KUKA KRL program: MyProgram_249().src

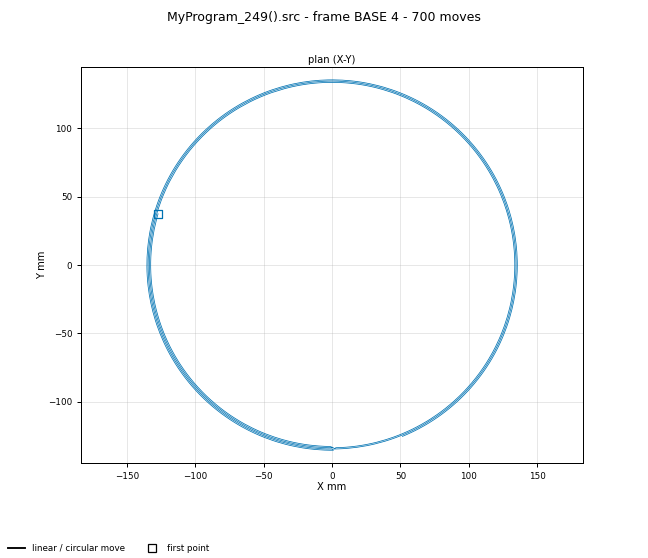
[picture p0: tool path of MyProgram_249().src in frame BASE 4, 700 of 700 moves have a stored position in this frame; points joined in program order, loops and branches not executed]
&ACCESS RVP
&REL 1
&PARAM TEMPLATE = C:\KRC\Roboter\Template\vorgabe
&PARAM EDITMASK = *
DEF MyProgram_249()
; ---- Setting reference (Base) ----
$BASE = BASE_DATA[4]

; --------------------------
; ---- Setting tool (TCP) ----
$TOOL = TOOL_DATA[3]
; --------------------------

$VEL.CP = VEL_APROX_PRINT
Startdeposition()
$VEL.CP = VEL_PRINT
LIN {X -127.2859,Y 37.4504,Z 164,A 163.9106,B 12.714,C 0.0045,E1 12.5602,E2 286.2896} C_DIS
LIN {X -128.1717,Y 34.2964,Z 164,A 165.3545,B 12.714,C 0.0079,E1 12.5591,E2 284.844} C_DIS
LIN {X -130.1138,Y 25.9783,Z 164,A 168.8195,B 12.714,C 0.0239,E1 12.557,E2 281.4101} C_DIS
LIN {X -131.4651,Y 17.9356,Z 164,A 172.8382,B 12.714,C 0.0228,E1 12.5551,E2 277.3369} C_DIS
LIN {X -131.9904,Y 13.5371,Z 164,A 174.6216,B 12.714,C 0.0315,E1 12.5546,E2 275.5713} C_DIS
LIN {X -132.3145,Y 9.8588,Z 164,A 176.2918,B 12.714,C 0.0344,E1 12.5542,E2 273.8938} C_DIS
LIN {X -132.5525,Y 5.8863,Z 164,A 178.0814,B 12.714,C 0.0379,E1 12.5539,E2 272.0978} C_DIS
LIN {X -132.6635,Y 2.1671,Z 164,A 179.6659,B 12.714,C 0.0432,E1 12.5539,E2 270.5176} C_DIS
LIN {X -132.6704,Y -1.7531,Z 164,A -178.5856,B 12.714,C 0.0469,E1 12.5539,E2 268.7644} C_DIS
LIN {X -132.5551,Y -5.8195,Z 164,A -176.8371,B 12.714,C 0.0523,E1 12.554,E2 267.0189} C_DIS
LIN {X -132.3464,Y -9.4225,Z 164,A -175.2437,B 12.714,C 0.0561,E1 12.5543,E2 265.423} C_DIS
LIN {X -132.026,Y -13.1779,Z 164,A -173.5549,B 12.7139,C 0.0595,E1 12.5548,E2 263.7286} C_DIS
LIN {X -131.5827,Y -17.0384,Z 164,A -171.2367,B 12.7139,C 0.0494,E1 12.5556,E2 261.3351} C_DIS
LIN {X -130.7769,Y -22.4052,Z 164,A -169.5669,B 12.7139,C 0.072,E1 12.5564,E2 259.749} C_DIS
LIN {X -129.5394,Y -28.7106,Z 164,A -166.6985,B 12.7138,C 0.0779,E1 12.558,E2 256.8722} C_DIS
LIN {X -128.5013,Y -33.0423,Z 164,A -164.2137,B 12.7138,C 0.0701,E1 12.5597,E2 254.3216} C_DIS
LIN {X -127.2066,Y -37.7213,Z 164,A -162.6596,B 12.7138,C 0.0888,E1 12.5609,E2 252.8349} C_DIS
LIN {X -125.9532,Y -41.7138,Z 164,A -160.9153,B 12.7137,C 0.0954,E1 12.5623,E2 251.0997} C_DIS
LIN {X -124.788,Y -45.0792,Z 164,A -159.3157,B 12.7137,C 0.0982,E1 12.5638,E2 249.4941} C_DIS
LIN {X -123.3299,Y -48.933,Z 164,A -157.4471,B 12.7137,C 0.1009,E1 12.5657,E2 247.6164} C_DIS
LIN {X -122.0827,Y -51.9667,Z 164,A -156.1315,B 12.7136,C 0.1071,E1 12.5671,E2 246.3141} C_DIS
LIN {X -120.6653,Y -55.1756,Z 164,A -154.4483,B 12.7136,C 0.1071,E1 12.5691,E2 244.6119} C_DIS
LIN {X -118.5377,Y -59.6103,Z 164,A -152.3885,B 12.7136,C 0.1142,E1 12.5716,E2 242.5616} C_DIS
LIN {X -116.8408,Y -62.8722,Z 164,A -150.792,B 12.7135,C 0.1181,E1 12.5737,E2 240.9653} C_DIS
LIN {X -114.9119,Y -66.3322,Z 164,A -148.9965,B 12.7135,C 0.1204,E1 12.5762,E2 239.1609} C_DIS
LIN {X -112.7429,Y -69.9553,Z 164,A -146.8726,B 12.7135,C 0.1177,E1 12.5793,E2 237.0019} C_DIS
LIN {X -110.8171,Y -72.9675,Z 164,A -145.2284,B 12.7135,C 0.119,E1 12.5819,E2 235.3465} C_DIS
LIN {X -108.5489,Y -76.3012,Z 164,A -143.8692,B 12.7133,C 0.1323,E1 12.584,E2 234.0348} C_DIS
LIN {X -106.1417,Y -79.6164,Z 164,A -142.0172,B 12.7133,C 0.1344,E1 12.5871,E2 232.1738} C_DIS
LIN {X -103.4343,Y -83.1029,Z 164,A -140.1059,B 12.7133,C 0.1386,E1 12.5904,E2 230.2631} C_DIS
LIN {X -101.023,Y -86.0177,Z 164,A -138.0843,B 12.7133,C 0.1327,E1 12.5941,E2 228.1952} C_DIS
LIN {X -98.2832,Y -89.135,Z 164,A -136.5931,B 12.7133,C 0.1438,E1 12.5968,E2 226.7415} C_DIS
LIN {X -95.0015,Y -92.6258,Z 164,A -134.5379,B 12.7132,C 0.1484,E1 12.6008,E2 224.6891} C_DIS
LIN {X -91.8567,Y -95.7449,Z 164,A -132.7035,B 12.7132,C 0.1541,E1 12.6044,E2 222.865} C_DIS
LIN {X -88.8171,Y -98.5716,Z 164,A -130.8078,B 12.7131,C 0.155,E1 12.6084,E2 220.9575} C_DIS
LIN {X -83.7542,Y -102.9072,Z 164,A -127.8819,B 12.7131,C 0.1591,E1 12.6147,E2 218.0268} C_DIS
LIN {X -80.3922,Y -105.5549,Z 164,A -126.3364,B 12.7129,C 0.1698,E1 12.618,E2 216.5186} C_DIS
LIN {X -77.3944,Y -107.7723,Z 164,A -124.7502,B 12.7129,C 0.173,E1 12.6215,E2 214.9358} C_DIS
LIN {X -74.3027,Y -109.9264,Z 164,A -122.8693,B 12.7129,C 0.1692,E1 12.6259,E2 213.0246} C_DIS
LIN {X -71.2377,Y -111.9375,Z 164,A -121.027,B 12.7129,C 0.1651,E1 12.6303,E2 211.151} C_DIS
LIN {X -66.9659,Y -114.544,Z 164,A -119.1475,B 12.7129,C 0.1752,E1 12.6348,E2 209.3062} C_DIS
LIN {X -63.868,Y -116.2999,Z 164,A -117.7538,B 12.7128,C 0.1809,E1 12.6381,E2 207.9301} C_DIS
LIN {X -60.867,Y -117.8979,Z 164,A -116.1634,B 12.7128,C 0.1797,E1 12.6421,E2 206.3251} C_DIS
LIN {X -58.2643,Y -119.2043,Z 164,A -114.7229,B 12.7128,C 0.1765,E1 12.6457,E2 204.8623} C_DIS
LIN {X -54.5493,Y -120.9492,Z 164,A -113.2139,B 12.7127,C 0.1852,E1 12.6495,E2 203.3854} C_DIS
LIN {X -51.4956,Y -122.2805,Z 164,A -111.5729,B 12.7127,C 0.1815,E1 12.6538,E2 201.7199} C_DIS
LIN {X -48.452,Y -123.5182,Z 164,A -110.1328,B 12.7127,C 0.1824,E1 12.6575,E2 200.2771} C_DIS
LIN {X -44.8785,Y -124.8604,Z 164,A -108.5366,B 12.7127,C 0.1852,E1 12.6617,E2 198.6871} C_DIS
LIN {X -42.0608,Y -125.8376,Z 164,A -107.0295,B 12.7127,C 0.1805,E1 12.6657,E2 197.1532} C_DIS
LIN {X -36.4597,Y -127.5753,Z 164,A -104.6656,B 12.7127,C 0.1868,E1 12.672,E2 194.8096} C_DIS
LIN {X -31.6264,Y -128.8576,Z 164,A -102.4818,B 12.7127,C 0.1874,E1 12.6779,E2 192.6224} C_DIS
LIN {X -27.87,Y -129.7209,Z 164,A -100.846,B 12.7127,C 0.189,E1 12.6824,E2 190.9897} C_DIS
LIN {X -23.7795,Y -130.5333,Z 164,A -99.0245,B 12.7127,C 0.1892,E1 12.6874,E2 189.1652} C_DIS
LIN {X -19.9907,Y -131.1668,Z 164,A -97.3285,B 12.7127,C 0.1888,E1 12.6921,E2 187.4642} C_DIS
LIN {X -16.2833,Y -131.6793,Z 164,A -95.708,B 12.7127,C 0.1891,E1 12.6966,E2 185.8426} C_DIS
LIN {X -12.7821,Y -132.064,Z 164,A -94.3224,B 12.7126,C 0.1929,E1 12.7004,E2 184.4731} C_DIS
LIN {X -9.6689,Y -132.3284,Z 164,A -92.921,B 12.7126,C 0.1917,E1 12.7043,E2 183.0647} C_DIS
LIN {X -5.4853,Y -132.5681,Z 164,A -91.0911,B 12.7126,C 0.1911,E1 12.7094,E2 181.2315} C_DIS
LIN {X -1.4506,Y -132.6753,Z 164,A -89.2488,B 12.7126,C 0.1883,E1 12.7146,E2 179.3764} C_DIS
LIN {X -1.4506,Y -132.6753,Z 164,A -89.2488,B 12.7126,C 0.1883,E1 12.7146,E2 179.3764} C_DIS
Enddeposition()
LIN {X 0.969,Y -133.5975,Z 164,A -88.8954,B 12.4309,C 0.2318,E1 12.434,E2 179.2272} C_DIS
Startdeposition()
$VEL.CP = VEL_PRINT
LIN {X -2.4265,Y -133.579,Z 164,A -90.4296,B 12.4309,C 0.2339,E1 12.4297,E2 180.7716} C_DIS
LIN {X -6.5842,Y -133.4385,Z 164,A -92.1314,B 12.4309,C 0.2318,E1 12.425,E2 182.4641} C_DIS
LIN {X -10.1796,Y -133.2132,Z 164,A -93.6549,B 12.4309,C 0.2312,E1 12.4207,E2 183.9856} C_DIS
LIN {X -14.0414,Y -132.8611,Z 164,A -95.3566,B 12.4309,C 0.2319,E1 12.416,E2 185.6927} C_DIS
LIN {X -17.9058,Y -132.3965,Z 164,A -97.0831,B 12.4309,C 0.233,E1 12.4112,E2 187.4267} C_DIS
LIN {X -21.716,Y -131.8242,Z 164,A -98.6443,B 12.4309,C 0.2301,E1 12.4069,E2 188.9773} C_DIS
LIN {X -24.9459,Y -131.2511,Z 164,A -100.0743,B 12.4309,C 0.2301,E1 12.403,E2 190.4105} C_DIS
LIN {X -28.3703,Y -130.5537,Z 164,A -101.5641,B 12.4309,C 0.2292,E1 12.3989,E2 191.8996} C_DIS
LIN {X -32.1236,Y -129.6833,Z 164,A -103.5588,B 12.4309,C 0.237,E1 12.3934,E2 193.9362} C_DIS
LIN {X -35.422,Y -128.8205,Z 164,A -104.7421,B 12.4309,C 0.229,E1 12.3903,E2 195.086} C_DIS
LIN {X -39.156,Y -127.7337,Z 164,A -106.311,B 12.431,C 0.2253,E1 12.3861,E2 196.643} C_DIS
LIN {X -42.2612,Y -126.7402,Z 164,A -107.7812,B 12.431,C 0.226,E1 12.3822,E2 198.1221} C_DIS
LIN {X -45.5289,Y -125.6035,Z 164,A -109.2648,B 12.431,C 0.2247,E1 12.3783,E2 199.6059} C_DIS
LIN {X -48.8747,Y -124.3406,Z 164,A -110.7775,B 12.431,C 0.2228,E1 12.3743,E2 201.1161} C_DIS
LIN {X -52.0639,Y -123.0398,Z 164,A -112.2452,B 12.4311,C 0.221,E1 12.3705,E2 202.5827} C_DIS
LIN {X -54.7996,Y -121.8447,Z 164,A -113.5516,B 12.4311,C 0.2203,E1 12.3672,E2 203.8922} C_DIS
LIN {X -58.0083,Y -120.3507,Z 164,A -115.2414,B 12.4311,C 0.2228,E1 12.3629,E2 205.6027} C_DIS
LIN {X -61.7986,Y -118.4487,Z 164,A -116.9737,B 12.4311,C 0.2184,E1 12.3586,E2 207.3245} C_DIS
LIN {X -65.64,Y -116.3658,Z 164,A -118.894,B 12.4311,C 0.2171,E1 12.3539,E2 209.2502} C_DIS
LIN {X -70.4553,Y -113.5145,Z 164,A -121.2134,B 12.4313,C 0.2118,E1 12.3484,E2 211.5595} C_DIS
LIN {X -73.3669,Y -111.6552,Z 164,A -122.786,B 12.4313,C 0.2118,E1 12.3447,E2 213.1428} C_DIS
LIN {X -77.4171,Y -108.8866,Z 164,A -124.79,B 12.4313,C 0.206,E1 12.3401,E2 215.1342} C_DIS
LIN {X -80.6674,Y -106.5007,Z 164,A -126.4,B 12.4315,C 0.2002,E1 12.3365,E2 216.7293} C_DIS
LIN {X -83.028,Y -104.6707,Z 164,A -128.3488,B 12.4312,C 0.2141,E1 12.3321,E2 218.7582} C_DIS
LIN {X -86.3499,Y -101.9476,Z 164,A -129.6511,B 12.4315,C 0.1979,E1 12.3294,E2 219.995} C_DIS
LIN {X -88.928,Y -99.7068,Z 164,A -131.2517,B 12.4315,C 0.1984,E1 12.326,E2 221.6115} C_DIS
LIN {X -92.0866,Y -96.7973,Z 164,A -133.0736,B 12.4315,C 0.1944,E1 12.3223,E2 223.4302} C_DIS
LIN {X -94.9521,Y -93.9879,Z 164,A -134.8716,B 12.4315,C 0.1927,E1 12.3187,E2 225.2367} C_DIS
LIN {X -97.949,Y -90.8604,Z 164,A -137.1822,B 12.4315,C 0.1996,E1 12.3142,E2 227.6007} C_DIS
LIN {X -100.953,Y -87.5114,Z 164,A -138.4296,B 12.4318,C 0.1794,E1 12.3121,E2 228.7653} C_DIS
LIN {X -102.7055,Y -85.4473,Z 164,A -139.8951,B 12.4318,C 0.184,E1 12.3094,E2 230.2669} C_DIS
LIN {X -105.5735,Y -81.8768,Z 164,A -141.7703,B 12.4318,C 0.1775,E1 12.3062,E2 232.1302} C_DIS
LIN {X -107.9313,Y -78.7438,Z 164,A -143.5646,B 12.4318,C 0.1763,E1 12.3032,E2 233.9371} C_DIS
LIN {X -110.9733,Y -74.3946,Z 164,A -145.7108,B 12.4319,C 0.1679,E1 12.2998,E2 236.0663} C_DIS
LIN {X -113.4173,Y -70.6123,Z 164,A -147.7572,B 12.4319,C 0.1658,E1 12.2967,E2 238.1251} C_DIS
LIN {X -115.5704,Y -67.0303,Z 164,A -149.5797,B 12.432,C 0.1621,E1 12.2941,E2 239.95} C_DIS
LIN {X -117.5621,Y -63.4729,Z 164,A -151.3707,B 12.432,C 0.1586,E1 12.2917,E2 241.7448} C_DIS
LIN {X -119.4403,Y -59.8644,Z 164,A -153.3097,B 12.432,C 0.1586,E1 12.2892,E2 243.7057} C_DIS
LIN {X -121.6776,Y -55.1732,Z 164,A -155.4943,B 12.4321,C 0.1517,E1 12.2866,E2 245.8832} C_DIS
LIN {X -123.4205,Y -51.1523,Z 164,A -157.1832,B 12.4322,C 0.1423,E1 12.2848,E2 247.5477} C_DIS
LIN {X -124.8044,Y -47.6815,Z 164,A -158.798,B 12.4322,C 0.1382,E1 12.2832,E2 249.1627} C_DIS
LIN {X -125.8056,Y -44.9683,Z 164,A -160.0935,B 12.4323,C 0.136,E1 12.2819,E2 250.4636} C_DIS
LIN {X -127.0792,Y -41.235,Z 164,A -161.8357,B 12.4323,C 0.1325,E1 12.2804,E2 252.2104} C_DIS
LIN {X -128.2024,Y -37.5929,Z 164,A -164.0108,B 12.4323,C 0.1402,E1 12.2786,E2 254.4481} C_DIS
LIN {X -129.4444,Y -33.0647,Z 164,A -165.5735,B 12.4324,C 0.1243,E1 12.2776,E2 255.9555} C_DIS
LIN {X -130.6401,Y -27.9703,Z 164,A -168.3192,B 12.4324,C 0.1291,E1 12.2759,E2 258.7584} C_DIS
LIN {X -131.5391,Y -23.3797,Z 164,A -169.7929,B 12.4326,C 0.1114,E1 12.2752,E2 260.1671} C_DIS
LIN {X -132.3855,Y -17.9896,Z 164,A -172.1913,B 12.4326,C 0.1059,E1 12.2742,E2 262.5701} C_DIS
LIN {X -132.8479,Y -14.1632,Z 164,A -173.8147,B 12.4326,C 0.1003,E1 12.2737,E2 264.1883} C_DIS
LIN {X -133.2229,Y -10.0464,Z 164,A -175.6612,B 12.4326,C 0.0968,E1 12.2732,E2 266.0417} C_DIS
LIN {X -133.4376,Y -6.6024,Z 164,A -177.1199,B 12.4327,C 0.0919,E1 12.273,E2 267.4962} C_DIS
LIN {X -133.5742,Y -2.7138,Z 164,A -178.874,B 12.4327,C 0.0889,E1 12.2729,E2 269.2587} C_DIS
LIN {X -133.5972,Y 1.0787,Z 164,A 179.4492,B 12.4327,C 0.0853,E1 12.2729,E2 270.9397} C_DIS
LIN {X -133.5003,Y 5.1826,Z 164,A 177.7929,B 12.4328,C 0.0777,E1 12.273,E2 272.5816} C_DIS
LIN {X -133.328,Y 8.5399,Z 164,A 176.3503,B 12.4328,C 0.0734,E1 12.2732,E2 274.0227} C_DIS
LIN {X -133.0541,Y 12.092,Z 164,A 174.658,B 12.4328,C 0.0726,E1 12.2736,E2 275.7329} C_DIS
LIN {X -132.6486,Y 15.9224,Z 164,A 173.0231,B 12.4328,C 0.0673,E1 12.2741,E2 277.3637} C_DIS
LIN {X -131.3055,Y 24.6614,Z 164,A 169.4185,B 12.4329,C 0.052,E1 12.2757,E2 280.9419} C_DIS
LIN {X -130.3282,Y 29.3907,Z 164,A 166.9317,B 12.4329,C 0.0553,E1 12.2772,E2 283.4754} C_DIS
LIN {X -129.1549,Y 34.1785,Z 164,A 164.9442,B 12.4329,C 0.0464,E1 12.2785,E2 285.4455} C_DIS
LIN {X -128.1565,Y 37.7498,Z 164,A 163.4061,B 12.4329,C 0.0406,E1 12.2797,E2 286.9755} C_DIS
LIN {X -127.1567,Y 40.9924,Z 164,A 161.9634,B 12.4329,C 0.0362,E1 12.2809,E2 288.415} C_DIS
LIN {X -126.1016,Y 44.1317,Z 164,A 160.5161,B 12.433,C 0.0328,E1 12.2822,E2 289.8638} C_DIS
LIN {X -124.9839,Y 47.204,Z 164,A 159.0732,B 12.433,C 0.0298,E1 12.2836,E2 291.3099} C_DIS
LIN {X -123.7939,Y 50.2418,Z 164,A 157.6003,B 12.433,C 0.0275,E1 12.2852,E2 292.7898} C_DIS
LIN {X -121.5872,Y 55.3731,Z 164,A 155.2739,B 12.433,C 0.0194,E1 12.2878,E2 295.1052} C_DIS
LIN {X -120.0819,Y 58.5641,Z 164,A 153.5082,B 12.433,C 0.021,E1 12.2899,E2 296.8989} C_DIS
LIN {X -118.5664,Y 61.5743,Z 164,A 152.1424,B 12.433,C 0.0154,E1 12.2917,E2 298.2536} C_DIS
LIN {X -115.5947,Y 66.9882,Z 164,A 149.6992,B 12.433,C 0.0038,E1 12.295,E2 300.6695} C_DIS
LIN {X -114.4253,Y 68.9671,Z 164,A 147.98,B 12.433,C 0.0179,E1 12.2976,E2 302.4736} C_DIS
LIN {X -111.8785,Y 73.0265,Z 164,A 146.4944,B 12.433,C -0.0003,E1 12.2997,E2 303.8902} C_DIS
LIN {X -109.7337,Y 76.2109,Z 164,A 144.6442,B 12.433,C 0.0003,E1 12.3027,E2 305.7623} C_DIS
LIN {X -106.848,Y 80.2072,Z 164,A 142.5669,B 12.433,C -0.0057,E1 12.3061,E2 307.8329} C_DIS
LIN {X -104.0301,Y 83.829,Z 164,A 140.6438,B 12.433,C -0.0114,E1 12.3094,E2 309.7484} C_DIS
LIN {X -101.3278,Y 87.0763,Z 164,A 138.79,B 12.433,C -0.0146,E1 12.3128,E2 311.6051} C_DIS
LIN {X -98.5378,Y 90.2216,Z 164,A 136.94,B 12.433,C -0.0176,E1 12.3162,E2 313.4587} C_DIS
LIN {X -95.3819,Y 93.5514,Z 164,A 135.009,B 12.433,C -0.0227,E1 12.3199,E2 315.3831} C_DIS
LIN {X -92.2253,Y 96.6647,Z 164,A 133.0772,B 12.433,C -0.026,E1 12.3238,E2 317.3164} C_DIS
LIN {X -88.9304,Y 99.7047,Z 164,A 131.14,B 12.433,C -0.0296,E1 12.3278,E2 319.2533} C_DIS
LIN {X -85.6216,Y 102.5603,Z 164,A 129.2397,B 12.433,C -0.0327,E1 12.3319,E2 321.1546} C_DIS
LIN {X -82.2236,Y 105.3043,Z 164,A 127.3172,B 12.433,C -0.0351,E1 12.3361,E2 323.0809} C_DIS
LIN {X -78.5614,Y 108.0635,Z 164,A 125.3608,B 12.433,C -0.039,E1 12.3405,E2 325.0341} C_DIS
LIN {X -74.9376,Y 110.6071,Z 164,A 123.4511,B 12.433,C -0.042,E1 12.3449,E2 326.9432} C_DIS
LIN {X -71.3158,Y 112.9762,Z 164,A 121.6079,B 12.433,C -0.0454,E1 12.3492,E2 328.7831} C_DIS
LIN {X -67.6566,Y 115.2049,Z 164,A 119.7538,B 12.433,C -0.0479,E1 12.3536,E2 330.6373} C_DIS
LIN {X -60.2805,Y 119.2285,Z 164,A 116.1931,B 12.433,C -0.0542,E1 12.3624,E2 334.1897} C_DIS
LIN {X -56.5162,Y 121.0587,Z 164,A 113.7895,B 12.433,C -0.042,E1 12.3686,E2 336.6628} C_DIS
LIN {X -52.0532,Y 123.0443,Z 164,A 112.3832,B 12.4329,C -0.0611,E1 12.372,E2 337.9868} C_DIS
LIN {X -48.3185,Y 124.5568,Z 164,A 110.4886,B 12.4329,C -0.0591,E1 12.377,E2 339.8996} C_DIS
LIN {X -44.2124,Y 126.0737,Z 164,A 108.5419,B 12.4329,C -0.0594,E1 12.3821,E2 341.853} C_DIS
LIN {X -34.5806,Y 129.0477,Z 164,A 104.5946,B 12.4329,C -0.0726,E1 12.3925,E2 345.7527} C_DIS
LIN {X -29.4838,Y 130.3069,Z 164,A 101.4239,B 12.4329,C -0.0517,E1 12.4014,E2 349.0296} C_DIS
LIN {X -24.4604,Y 131.3439,Z 164,A 99.9031,B 12.4329,C -0.0697,E1 12.4054,E2 350.4697} C_DIS
LIN {X -21.7381,Y 131.8205,Z 164,A 98.642,B 12.4329,C -0.0685,E1 12.4089,E2 351.7389} C_DIS
LIN {X -17.7944,Y 132.4111,Z 164,A 96.9364,B 12.4329,C -0.0695,E1 12.4136,E2 353.443} C_DIS
LIN {X -14.2596,Y 132.8376,Z 164,A 95.4026,B 12.4329,C -0.0699,E1 12.4178,E2 354.9767} C_DIS
LIN {X -9.9853,Y 133.2274,Z 164,A 93.5465,B 12.4329,C -0.0701,E1 12.423,E2 356.8335} C_DIS
LIN {X -5.909,Y 133.472,Z 164,A 91.7239,B 12.4329,C -0.0687,E1 12.4281,E2 358.6637} C_DIS
LIN {X -2.1617,Y 133.5834,Z 164,A 90.2016,B 12.4329,C -0.0711,E1 12.4323,E2 360.1751} C_DIS
LIN {X 1.581,Y 133.5931,Z 164,A 88.5163,B 12.4329,C -0.0691,E1 12.437,E2 361.8691} C_DIS
LIN {X 5.7626,Y 133.4777,Z 164,A 86.718,B 12.4329,C -0.0689,E1 12.4421,E2 363.6671} C_DIS
LIN {X 9.8231,Y 133.2392,Z 164,A 85.0497,B 12.4329,C -0.0706,E1 12.4467,E2 365.3257} C_DIS
LIN {X 14.1296,Y 132.8516,Z 164,A 83.2116,B 12.4329,C -0.0706,E1 12.4518,E2 367.1613} C_DIS
LIN {X 18.068,Y 132.3752,Z 164,A 81.4185,B 12.4329,C -0.0677,E1 12.4568,E2 368.9647} C_DIS
LIN {X 21.7746,Y 131.8144,Z 164,A 79.8952,B 12.4329,C -0.0693,E1 12.461,E2 370.4775} C_DIS
LIN {X 25.3119,Y 131.1811,Z 164,A 78.3962,B 12.4329,C -0.0697,E1 12.4651,E2 371.9712} C_DIS
LIN {X 29.0207,Y 130.4127,Z 164,A 76.4019,B 12.4329,C -0.0591,E1 12.4706,E2 374.0088} C_DIS
LIN {X 32.4462,Y 129.6014,Z 164,A 75.4247,B 12.4329,C -0.0721,E1 12.4731,E2 374.9228} C_DIS
LIN {X 37.1312,Y 128.3376,Z 164,A 73.0542,B 12.4329,C -0.0629,E1 12.4796,E2 377.3272} C_DIS
LIN {X 41.1205,Y 127.1158,Z 164,A 71.524,B 12.4329,C -0.0683,E1 12.4836,E2 378.8265} C_DIS
LIN {X 43.8424,Y 126.2019,Z 164,A 70.2132,B 12.4329,C -0.0651,E1 12.4871,E2 380.1466} C_DIS
LIN {X 46.7073,Y 125.17,Z 164,A 68.8618,B 12.4329,C -0.0627,E1 12.4906,E2 381.5034} C_DIS
LIN {X 49.9839,Y 123.8978,Z 164,A 67.3652,B 12.4329,C -0.0614,E1 12.4945,E2 382.9986} C_DIS
LIN {X 53.78,Y 122.3006,Z 164,A 65.5905,B 12.4329,C -0.0592,E1 12.4991,E2 384.7744} C_DIS
LIN {X 57.2668,Y 120.7049,Z 164,A 64.1702,B 12.4329,C -0.0633,E1 12.5026,E2 386.1681} C_DIS
LIN {X 59.8901,Y 119.4264,Z 164,A 62.6216,B 12.4329,C -0.0537,E1 12.5066,E2 387.7521} C_DIS
LIN {X 64.0154,Y 117.2672,Z 164,A 60.4917,B 12.4329,C -0.0474,E1 12.5118,E2 389.8979} C_DIS
LIN {X 68.7061,Y 114.5826,Z 164,A 58.3496,B 12.4329,C -0.0489,E1 12.5169,E2 392.0197} C_DIS
LIN {X 72.3757,Y 112.3009,Z 164,A 56.3459,B 12.4329,C -0.0419,E1 12.5217,E2 394.0416} C_DIS
LIN {X 76.7579,Y 109.3521,Z 164,A 54.2838,B 12.4329,C -0.0438,E1 12.5264,E2 396.0801} C_DIS
LIN {X 80.2832,Y 106.7906,Z 164,A 52.38,B 12.4329,C -0.0397,E1 12.5307,E2 397.9885} C_DIS
LIN {X 83.9771,Y 103.9107,Z 164,A 50.4288,B 12.4329,C -0.0377,E1 12.5349,E2 399.9335} C_DIS
LIN {X 87.3119,Y 101.1248,Z 164,A 48.5679,B 12.4329,C -0.0343,E1 12.5389,E2 401.7948} C_DIS
LIN {X 90.6735,Y 98.1224,Z 164,A 46.6797,B 12.433,C -0.0318,E1 12.5428,E2 403.6784} C_DIS
LIN {X 93.8368,Y 95.102,Z 164,A 44.7631,B 12.433,C -0.0269,E1 12.5467,E2 405.6008} C_DIS
LIN {X 96.9682,Y 91.9067,Z 164,A 42.859,B 12.433,C -0.0233,E1 12.5504,E2 407.504} C_DIS
LIN {X 99.9862,Y 88.6134,Z 164,A 40.9853,B 12.433,C -0.0203,E1 12.5538,E2 409.3737} C_DIS
LIN {X 102.9393,Y 85.165,Z 164,A 39.0707,B 12.433,C -0.0169,E1 12.5573,E2 411.2854} C_DIS
LIN {X 105.7218,Y 81.6854,Z 164,A 37.1508,B 12.433,C -0.0123,E1 12.5606,E2 413.2075} C_DIS
LIN {X 108.2126,Y 78.3556,Z 164,A 35.4604,B 12.433,C -0.0108,E1 12.5634,E2 414.8879} C_DIS
LIN {X 110.6534,Y 74.8691,Z 164,A 33.7908,B 12.433,C -0.0108,E1 12.566,E2 416.5399} C_DIS
LIN {X 112.5195,Y 72.0343,Z 164,A 32.1577,B 12.433,C -0.0022,E1 12.5685,E2 418.1953} C_DIS
LIN {X 114.9391,Y 68.108,Z 164,A 29.4929,B 12.433,C 0.0221,E1 12.5725,E2 420.9433} C_DIS
LIN {X 117.8168,Y 62.9988,Z 164,A 27.9523,B 12.433,C 0.001,E1 12.5744,E2 422.3695} C_DIS
LIN {X 120.5626,Y 57.5646,Z 164,A 25.2218,B 12.433,C 0.0112,E1 12.5778,E2 425.1165} C_DIS
LIN {X 121.9199,Y 54.6314,Z 164,A 23.7886,B 12.433,C 0.0162,E1 12.5795,E2 426.5565} C_DIS
LIN {X 123.3732,Y 51.2656,Z 164,A 22.2535,B 12.433,C 0.0194,E1 12.5811,E2 428.0885} C_DIS
LIN {X 124.6316,Y 48.1259,Z 164,A 20.7955,B 12.433,C 0.0236,E1 12.5826,E2 429.5485} C_DIS
LIN {X 125.7505,Y 45.1213,Z 164,A 19.4725,B 12.433,C 0.0259,E1 12.5839,E2 430.8665} C_DIS
LIN {X 127.4742,Y 39.9946,Z 164,A 16.9407,B 12.433,C 0.0385,E1 12.5861,E2 433.4259} C_DIS
LIN {X 129.3411,Y 33.4721,Z 164,A 14.408,B 12.433,C 0.0359,E1 12.588,E2 435.916} C_DIS
LIN {X 130.3362,Y 29.3557,Z 164,A 12.5555,B 12.433,C 0.0421,E1 12.5892,E2 437.7747} C_DIS
LIN {X 131.1214,Y 25.6242,Z 164,A 10.8378,B 12.433,C 0.0492,E1 12.5901,E2 439.5039} C_DIS
LIN {X 131.8393,Y 21.6254,Z 164,A 9.2398,B 12.433,C 0.0501,E1 12.5909,E2 441.0862} C_DIS
LIN {X 132.3325,Y 18.3723,Z 164,A 7.7932,B 12.433,C 0.0552,E1 12.5915,E2 442.5386} C_DIS
LIN {X 132.8163,Y 14.4577,Z 164,A 6.1079,B 12.433,C 0.06,E1 12.592,E2 444.2248} C_DIS
LIN {X 133.1793,Y 10.6221,Z 164,A 4.5234,B 12.4329,C 0.0629,E1 12.5924,E2 445.803} C_DIS
LIN {X 133.4272,Y 6.8099,Z 164,A 2.8724,B 12.4329,C 0.0681,E1 12.5927,E2 447.4572} C_DIS
LIN {X 133.5574,Y 3.4183,Z 164,A 1.4395,B 12.4329,C 0.0718,E1 12.5928,E2 448.8889} C_DIS
LIN {X 133.6005,Y -0.45,Z 164,A -0.2817,B 12.4328,C 0.0785,E1 12.5928,E2 450.6195} C_DIS
LIN {X 133.5338,Y -4.2679,Z 164,A -1.8077,B 12.4328,C 0.0801,E1 12.5928,E2 452.1339} C_DIS
LIN {X 133.3642,Y -7.9518,Z 164,A -3.4191,B 12.4328,C 0.0857,E1 12.5925,E2 453.7506} C_DIS
LIN {X 133.0955,Y -11.6138,Z 164,A -5.0672,B 12.4328,C 0.0925,E1 12.5921,E2 455.4094} C_DIS
LIN {X 132.6764,Y -15.6891,Z 164,A -6.7244,B 12.4327,C 0.0948,E1 12.5916,E2 457.0565} C_DIS
LIN {X 132.0952,Y -20.0046,Z 164,A -8.6204,B 12.4327,C 0.1011,E1 12.5909,E2 458.9582} C_DIS
LIN {X 131.4166,Y -24.0642,Z 164,A -10.2184,B 12.4327,C 0.1015,E1 12.5901,E2 460.5379} C_DIS
LIN {X 130.8487,Y -26.9788,Z 164,A -11.6383,B 12.4326,C 0.1095,E1 12.5893,E2 461.9771} C_DIS
LIN {X 129.8999,Y -31.2271,Z 164,A -14.3392,B 12.4323,C 0.139,E1 12.5875,E2 464.7806} C_DIS
LIN {X 128.1272,Y -37.85,Z 164,A -16.2643,B 12.4325,C 0.1182,E1 12.5861,E2 466.587} C_DIS
LIN {X 125.9578,Y -44.5462,Z 164,A -19.2429,B 12.4325,C 0.1256,E1 12.5835,E2 469.5644} C_DIS
LIN {X 124.739,Y -47.8497,Z 164,A -20.6532,B 12.4325,C 0.127,E1 12.5821,E2 470.9643} C_DIS
LIN {X 123.8122,Y -50.1962,Z 164,A -21.8575,B 12.4323,C 0.1335,E1 12.5809,E2 472.1848} C_DIS
LIN {X 122.326,Y -53.7212,Z 164,A -23.5009,B 12.4323,C 0.1382,E1 12.579,E2 473.8307} C_DIS
LIN {X 119.61,Y -59.5206,Z 164,A -26.2639,B 12.4322,C 0.1462,E1 12.5757,E2 476.599} C_DIS
LIN {X 117.5175,Y -63.5558,Z 164,A -28.2114,B 12.4322,C 0.1513,E1 12.5732,E2 478.5486} C_DIS
LIN {X 114.6621,Y -68.5727,Z 164,A -30.4171,B 12.4322,C 0.1501,E1 12.5701,E2 480.7243} C_DIS
LIN {X 112.8828,Y -71.4638,Z 164,A -32.0436,B 12.432,C 0.1587,E1 12.5677,E2 482.3735} C_DIS
LIN {X 110.4275,Y -75.2029,Z 164,A -33.9648,B 12.432,C 0.1637,E1 12.5647,E2 484.2973} C_DIS
LIN {X 107.8888,Y -78.8017,Z 164,A -35.8754,B 12.432,C 0.169,E1 12.5616,E2 486.2127} C_DIS
LIN {X 105.1322,Y -82.4427,Z 164,A -37.7572,B 12.4319,C 0.1716,E1 12.5584,E2 488.0874} C_DIS
LIN {X 102.4381,Y -85.7672,Z 164,A -39.667,B 12.4318,C 0.178,E1 12.555,E2 490.0085} C_DIS
LIN {X 99.015,Y -89.6973,Z 164,A -41.6276,B 12.4318,C 0.1754,E1 12.5514,E2 491.9381} C_DIS
LIN {X 96.5864,Y -92.3073,Z 164,A -43.858,B 12.4315,C 0.1987,E1 12.547,E2 494.2556} C_DIS
LIN {X 93.0399,Y -95.881,Z 164,A -45.3331,B 12.4317,C 0.184,E1 12.5442,E2 495.6499} C_DIS
LIN {X 89.2122,Y -99.4523,Z 164,A -47.3632,B 12.4317,C 0.1827,E1 12.5401,E2 497.6563} C_DIS
LIN {X 87.0244,Y -101.3724,Z 164,A -49.4614,B 12.4313,C 0.2092,E1 12.5354,E2 499.8594} C_DIS
LIN {X 83.1556,Y -104.5692,Z 164,A -51.3716,B 12.4313,C 0.2066,E1 12.5313,E2 501.7426} C_DIS
LIN {X 80.0873,Y -106.938,Z 164,A -52.5838,B 12.4315,C 0.1971,E1 12.5287,E2 502.9017} C_DIS
LIN {X 77.1157,Y -109.0997,Z 164,A -54.1973,B 12.4315,C 0.2011,E1 12.525,E2 504.5214} C_DIS
LIN {X 72.309,Y -112.3426,Z 164,A -56.7467,B 12.4313,C 0.2072,E1 12.5191,E2 507.081} C_DIS
LIN {X 69.3795,Y -114.1759,Z 164,A -58.2352,B 12.4313,C 0.2099,E1 12.5155,E2 508.5718} C_DIS
LIN {X 65.4087,Y -116.4958,Z 164,A -60.1255,B 12.4313,C 0.2107,E1 12.511,E2 510.454} C_DIS
LIN {X 61.7499,Y -118.4742,Z 164,A -61.8687,B 12.4313,C 0.2123,E1 12.5067,E2 512.1939} C_DIS
LIN {X 58.8357,Y -119.9479,Z 164,A -63.2454,B 12.4313,C 0.2136,E1 12.5033,E2 513.5689} C_DIS
LIN {X 55.6551,Y -121.4569,Z 164,A -64.797,B 12.4312,C 0.2169,E1 12.4993,E2 515.1271} C_DIS
LIN {X 51.6811,Y -123.1997,Z 164,A -66.6162,B 12.4312,C 0.2181,E1 12.4947,E2 516.9427} C_DIS
LIN {X 48.45,Y -124.5057,Z 164,A -68.1035,B 12.4312,C 0.2198,E1 12.4908,E2 518.4304} C_DIS
LIN {X 44.5996,Y -125.9386,Z 164,A -70.5964,B 12.4307,C 0.2417,E1 12.484,E2 521.0137} C_DIS
LIN {X 39.2866,Y -127.6937,Z 164,A -72.0183,B 12.4312,C 0.2176,E1 12.4805,E2 522.3185} C_DIS
LIN {X 32.6398,Y -129.5523,Z 164,A -75.0709,B 12.4311,C 0.2229,E1 12.4723,E2 525.3849} C_DIS
LIN {X 29.5894,Y -130.2828,Z 164,A -76.5052,B 12.4311,C 0.2264,E1 12.4683,E2 526.8311} C_DIS
LIN {X 25.7108,Y -131.1048,Z 164,A -78.3466,B 12.4309,C 0.2314,E1 12.4632,E2 528.6909} C_DIS
LIN {X 21.9613,Y -131.7833,Z 164,A -79.8517,B 12.4309,C 0.229,E1 12.4591,E2 530.1813} C_DIS
LIN {X 17.977,Y -132.3872,Z 164,A -81.6334,B 12.4309,C 0.2314,E1 12.4542,E2 531.9707} C_DIS
LIN {X 14.2772,Y -132.8357,Z 164,A -83.1851,B 12.4309,C 0.2309,E1 12.4499,E2 533.5177} C_DIS
LIN {X 10.0727,Y -133.221,Z 164,A -85.0148,B 12.4309,C 0.2321,E1 12.4448,E2 535.3507} C_DIS
LIN {X 6.4839,Y -133.4436,Z 164,A -86.5022,B 12.4309,C 0.2311,E1 12.4407,E2 536.8323} C_DIS
LIN {X 2.8668,Y -133.5717,Z 164,A -88.1288,B 12.4309,C 0.2335,E1 12.4361,E2 538.4687} C_DIS
LIN {X 2.8668,Y -133.5717,Z 164,A -88.1288,B 12.4309,C 0.2335,E1 12.4361,E2 538.4687} C_DIS
Enddeposition()
LIN {X 0.9773,Y -134.5138,Z 164,A -88.3977,B 12.3544,C 0.2314,E1 12.3588,E2 538.7297} C_DIS
Startdeposition()
$VEL.CP = VEL_PRINT
LIN {X 3.736,Y -134.4686,Z 164,A -86.9565,B 12.3544,C 0.2241,E1 12.3629,E2 537.255} C_DIS
LIN {X 7.9797,Y -134.2839,Z 164,A -85.1298,B 12.3545,C 0.2231,E1 12.368,E2 535.4252} C_DIS
LIN {X 11.9741,Y -133.988,Z 164,A -83.5132,B 12.3545,C 0.2248,E1 12.3725,E2 533.8188} C_DIS
LIN {X 15.6479,Y -133.6075,Z 164,A -81.9269,B 12.3545,C 0.2237,E1 12.3769,E2 532.2299} C_DIS
LIN {X 18.4953,Y -133.2439,Z 164,A -80.6123,B 12.3545,C 0.2206,E1 12.3806,E2 530.903} C_DIS
LIN {X 22.1538,Y -132.6835,Z 164,A -79.1456,B 12.3545,C 0.2226,E1 12.3846,E2 529.449} C_DIS
LIN {X 25.1781,Y -132.143,Z 164,A -77.9599,B 12.3545,C 0.2251,E1 12.3878,E2 528.2777} C_DIS
LIN {X 27.4741,Y -131.6864,Z 164,A -76.8537,B 12.3545,C 0.2214,E1 12.3909,E2 527.1573} C_DIS
LIN {X 31.0953,Y -130.8776,Z 164,A -75.2449,B 12.3545,C 0.2194,E1 12.3953,E2 525.5437} C_DIS
LIN {X 36.0954,Y -129.5871,Z 164,A -73.3236,B 12.3545,C 0.225,E1 12.4004,E2 523.6555} C_DIS
LIN {X 38.6981,Y -128.8356,Z 164,A -71.3995,B 12.3549,C 0.2026,E1 12.4058,E2 521.6343} C_DIS
LIN {X 42.792,Y -127.5327,Z 164,A -69.8634,B 12.3548,C 0.2088,E1 12.4098,E2 520.1335} C_DIS
LIN {X 47.0229,Y -126.0338,Z 164,A -68.1758,B 12.3547,C 0.2129,E1 12.4141,E2 518.4724} C_DIS
LIN {X 49.9546,Y -124.9012,Z 164,A -66.9174,B 12.3547,C 0.2135,E1 12.4174,E2 517.2229} C_DIS
LIN {X 52.5489,Y -123.8339,Z 164,A -65.4898,B 12.3548,C 0.2055,E1 12.4211,E2 515.7652} C_DIS
LIN {X 57.3346,Y -121.6918,Z 164,A -63.4877,B 12.3548,C 0.209,E1 12.4261,E2 513.79} C_DIS
LIN {X 60.6826,Y -120.0557,Z 164,A -61.8586,B 12.3548,C 0.2055,E1 12.4302,E2 512.1541} C_DIS
LIN {X 64.0533,Y -118.2941,Z 164,A -60.1207,B 12.3549,C 0.1997,E1 12.4346,E2 510.4} C_DIS
LIN {X 68.0375,Y -116.0477,Z 164,A -58.2278,B 12.3549,C 0.1982,E1 12.4391,E2 508.5121} C_DIS
LIN {X 75.4671,Y -111.3588,Z 164,A -54.4731,B 12.355,C 0.1914,E1 12.448,E2 504.7523} C_DIS
LIN {X 79.1479,Y -108.7741,Z 164,A -52.0684,B 12.3553,C 0.1739,E1 12.4535,E2 502.2842} C_DIS
LIN {X 83.1761,Y -105.7255,Z 164,A -49.9569,B 12.3553,C 0.1709,E1 12.4582,E2 500.1755} C_DIS
LIN {X 87.0037,Y -102.5989,Z 164,A -48.5275,B 12.3551,C 0.1861,E1 12.4611,E2 498.8286} C_DIS
LIN {X 93.0276,Y -97.17,Z 164,A -45.2416,B 12.3551,C 0.1838,E1 12.4678,E2 495.56} C_DIS
LIN {X 97.6517,Y -92.5223,Z 164,A -42.3377,B 12.3553,C 0.1745,E1 12.4735,E2 492.6393} C_DIS
LIN {X 102.2173,Y -87.4524,Z 164,A -39.3146,B 12.3554,C 0.1644,E1 12.4792,E2 489.5985} C_DIS
LIN {X 104.924,Y -84.1856,Z 164,A -37.5034,B 12.3554,C 0.16,E1 12.4824,E2 487.7847} C_DIS
LIN {X 107.6656,Y -80.6499,Z 164,A -35.6399,B 12.3555,C 0.1566,E1 12.4855,E2 485.9242} C_DIS
LIN {X 110.1299,Y -77.2508,Z 164,A -33.8705,B 12.3555,C 0.1527,E1 12.4884,E2 484.1551} C_DIS
LIN {X 112.5277,Y -73.714,Z 164,A -32.0969,B 12.3556,C 0.1494,E1 12.4911,E2 482.385} C_DIS
LIN {X 114.8393,Y -70.0586,Z 164,A -30.1345,B 12.3556,C 0.1411,E1 12.494,E2 480.4054} C_DIS
LIN {X 117.2056,Y -66.0229,Z 164,A -28.2751,B 12.3557,C 0.1398,E1 12.4966,E2 478.5602} C_DIS
LIN {X 119.2608,Y -62.2301,Z 164,A -26.4198,B 12.3557,C 0.1343,E1 12.499,E2 476.7004} C_DIS
LIN {X 120.9423,Y -58.8985,Z 164,A -25.0013,B 12.3557,C 0.1351,E1 12.5008,E2 475.3014} C_DIS
LIN {X 122.4278,Y -55.7465,Z 164,A -23.3555,B 12.3559,C 0.1262,E1 12.5027,E2 473.6337} C_DIS
LIN {X 124.0502,Y -52.0308,Z 164,A -21.8165,B 12.3559,C 0.127,E1 12.5044,E2 472.1159} C_DIS
LIN {X 125.1398,Y -49.3568,Z 164,A -20.3458,B 12.3559,C 0.1164,E1 12.5059,E2 470.6138} C_DIS
LIN {X 126.6986,Y -45.2028,Z 164,A -18.6702,B 12.3559,C 0.1174,E1 12.5075,E2 468.9626} C_DIS
LIN {X 128.0135,Y -41.3325,Z 164,A -16.9093,B 12.3559,C 0.1119,E1 12.5091,E2 467.1971} C_DIS
LIN {X 129.1142,Y -37.7517,Z 164,A -15.6253,B 12.3559,C 0.1165,E1 12.5101,E2 465.9499} C_DIS
LIN {X 130.5006,Y -32.6417,Z 164,A -13.105,B 12.3561,C 0.1021,E1 12.5119,E2 463.3941} C_DIS
LIN {X 131.3865,Y -28.8707,Z 164,A -11.5034,B 12.3561,C 0.0987,E1 12.5129,E2 461.7966} C_DIS
LIN {X 132.0307,Y -25.7654,Z 164,A -10.3526,B 12.3561,C 0.1007,E1 12.5135,E2 460.669} C_DIS
LIN {X 132.6518,Y -22.344,Z 164,A -8.7175,B 12.3561,C 0.0918,E1 12.5143,E2 459.013} C_DIS
LIN {X 133.2479,Y -18.4673,Z 164,A -6.9803,B 12.3562,C 0.0849,E1 12.515,E2 457.2657} C_DIS
LIN {X 133.7463,Y -14.4106,Z 164,A -5.393,B 12.3562,C 0.0843,E1 12.5155,E2 455.6954} C_DIS
LIN {X 134.0977,Y -10.6756,Z 164,A -3.8472,B 12.3562,C 0.0811,E1 12.5159,E2 454.1542} C_DIS
LIN {X 134.3388,Y -6.992,Z 164,A -2.1943,B 12.3562,C 0.074,E1 12.5161,E2 452.4896} C_DIS
LIN {X 134.4968,Y -2.5444,Z 164,A -0.3593,B 12.3562,C 0.0702,E1 12.5163,E2 450.66} C_DIS
LIN {X 134.5152,Y 1.3658,Z 164,A 1.2656,B 12.3563,C 0.0665,E1 12.5163,E2 449.0382} C_DIS
LIN {X 134.4306,Y 4.9264,Z 164,A 2.8378,B 12.3563,C 0.0603,E1 12.5161,E2 447.4575} C_DIS
LIN {X 134.1873,Y 9.467,Z 164,A 4.6903,B 12.3563,C 0.0571,E1 12.5158,E2 445.6134} C_DIS
LIN {X 133.8715,Y 13.2018,Z 164,A 6.3351,B 12.3563,C 0.051,E1 12.5154,E2 443.961} C_DIS
LIN {X 133.4456,Y 16.9778,Z 164,A 7.7151,B 12.3563,C 0.0533,E1 12.5149,E2 442.6088} C_DIS
LIN {X 132.9678,Y 20.3796,Z 164,A 9.3017,B 12.3564,C 0.0454,E1 12.5143,E2 441.0053} C_DIS
LIN {X 132.401,Y 23.7839,Z 164,A 10.71,B 12.3564,C 0.0429,E1 12.5136,E2 439.6031} C_DIS
LIN {X 131.7921,Y 26.9547,Z 164,A 12.1199,B 12.3564,C 0.0379,E1 12.5129,E2 438.1877} C_DIS
LIN {X 130.912,Y 30.9525,Z 164,A 13.8168,B 12.3564,C 0.0343,E1 12.5118,E2 436.4949} C_DIS
LIN {X 130.2151,Y 33.7667,Z 164,A 15.2604,B 12.3564,C 0.0246,E1 12.5108,E2 435.0244} C_DIS
LIN {X 127.3906,Y 43.2187,Z 164,A 19.2436,B 12.3564,C 0.0193,E1 12.5075,E2 431.0645} C_DIS
LIN {X 125.8844,Y 47.4218,Z 164,A 21.1552,B 12.3564,C 0.0138,E1 12.5057,E2 429.15} C_DIS
LIN {X 124.4008,Y 51.1913,Z 164,A 22.765,B 12.3564,C 0.0125,E1 12.504,E2 427.553} C_DIS
LIN {X 122.9569,Y 54.5653,Z 164,A 24.3588,B 12.3564,C 0.0074,E1 12.5022,E2 425.9541} C_DIS
LIN {X 121.5536,Y 57.6237,Z 164,A 25.9112,B 12.3564,C 0.0001,E1 12.5004,E2 424.3859} C_DIS
LIN {X 119.3042,Y 62.1474,Z 164,A 27.9233,B 12.3564,C -0.0014,E1 12.4979,E2 422.3894} C_DIS
LIN {X 117.6215,Y 65.2789,Z 164,A 29.578,B 12.3564,C -0.0094,E1 12.4956,E2 420.7163} C_DIS
LIN {X 115.1623,Y 69.5256,Z 164,A 31.5251,B 12.3564,C -0.0105,E1 12.4929,E2 418.7853} C_DIS
LIN {X 112.7993,Y 73.2971,Z 164,A 33.3559,B 12.3564,C -0.0133,E1 12.4901,E2 416.9612} C_DIS
LIN {X 110.8731,Y 76.1794,Z 164,A 34.8079,B 12.3564,C -0.0161,E1 12.4878,E2 415.5112} C_DIS
LIN {X 108.3389,Y 79.7423,Z 164,A 36.7321,B 12.3564,C -0.0223,E1 12.4847,E2 413.5783} C_DIS
LIN {X 105.7141,Y 83.1907,Z 164,A 38.5276,B 12.3564,C -0.0251,E1 12.4816,E2 411.7879} C_DIS
LIN {X 103.035,Y 86.4866,Z 164,A 40.3357,B 12.3564,C -0.0291,E1 12.4784,E2 409.9789} C_DIS
LIN {X 100.1741,Y 89.7848,Z 164,A 42.1595,B 12.3564,C -0.0321,E1 12.475,E2 408.1586} C_DIS
LIN {X 97.0931,Y 93.1081,Z 164,A 44.0703,B 12.3564,C -0.0356,E1 12.4714,E2 406.2493} C_DIS
LIN {X 93.9503,Y 96.2787,Z 164,A 45.9985,B 12.3564,C -0.0402,E1 12.4675,E2 404.3169} C_DIS
LIN {X 90.6581,Y 99.385,Z 164,A 47.9282,B 12.3564,C -0.0441,E1 12.4636,E2 402.3862} C_DIS
LIN {X 87.3123,Y 102.3366,Z 164,A 49.7718,B 12.3564,C -0.0461,E1 12.4597,E2 400.5488} C_DIS
LIN {X 84.0449,Y 105.0368,Z 164,A 51.5975,B 12.3564,C -0.0499,E1 12.4558,E2 398.7201} C_DIS
LIN {X 80.6919,Y 107.6343,Z 164,A 53.3979,B 12.3564,C -0.0528,E1 12.4518,E2 396.92} C_DIS
LIN {X 77.4063,Y 110.0201,Z 164,A 55.0331,B 12.3564,C -0.0531,E1 12.4481,E2 395.2957} C_DIS
LIN {X 73.8133,Y 112.4624,Z 164,A 56.9017,B 12.3564,C -0.0565,E1 12.4437,E2 393.4246} C_DIS
LIN {X 70.0255,Y 114.8596,Z 164,A 58.5571,B 12.3564,C -0.0524,E1 12.4399,E2 391.7996} C_DIS
LIN {X 64.1356,Y 118.2492,Z 164,A 61.4262,B 12.3564,C -0.0557,E1 12.4329,E2 388.9333} C_DIS
LIN {X 61.0495,Y 119.869,Z 164,A 62.9963,B 12.3564,C -0.06,E1 12.429,E2 387.3527} C_DIS
LIN {X 58.6333,Y 121.0713,Z 164,A 64.3557,B 12.3564,C -0.0672,E1 12.4255,E2 385.9679} C_DIS
LIN {X 55.1148,Y 122.7111,Z 164,A 65.8636,B 12.3564,C -0.0652,E1 12.4217,E2 384.4775} C_DIS
LIN {X 52.0456,Y 124.0441,Z 164,A 67.1656,B 12.3564,C -0.0634,E1 12.4184,E2 383.1904} C_DIS
LIN {X 49.5474,Y 125.0653,Z 164,A 68.5974,B 12.3563,C -0.0722,E1 12.4146,E2 381.7246} C_DIS
LIN {X 45.6734,Y 126.529,Z 164,A 70.1287,B 12.3563,C -0.0677,E1 12.4107,E2 380.2214} C_DIS
LIN {X 43.0805,Y 127.4366,Z 164,A 71.4412,B 12.3563,C -0.0725,E1 12.4072,E2 378.8918} C_DIS
LIN {X 39.2505,Y 128.6665,Z 164,A 73.1266,B 12.3563,C -0.0732,E1 12.4027,E2 377.21} C_DIS
LIN {X 34.8815,Y 129.9192,Z 164,A 74.9501,B 12.3563,C -0.0716,E1 12.3978,E2 375.4004} C_DIS
LIN {X 31.73,Y 130.7246,Z 164,A 76.4524,B 12.3563,C -0.0756,E1 12.3937,E2 373.8842} C_DIS
LIN {X 27.3077,Y 131.7203,Z 164,A 78.3473,B 12.3563,C -0.0757,E1 12.3886,E2 371.9941} C_DIS
LIN {X 23.7872,Y 132.4005,Z 164,A 79.7962,B 12.3563,C -0.0744,E1 12.3846,E2 370.5551} C_DIS
LIN {X 20.9446,Y 132.8803,Z 164,A 80.9217,B 12.3563,C -0.0722,E1 12.3815,E2 369.4422} C_DIS
LIN {X 18.1899,Y 133.2868,Z 164,A 82.3306,B 12.3563,C -0.0785,E1 12.3776,E2 368.0069} C_DIS
LIN {X 14.6644,Y 133.719,Z 164,A 83.7836,B 12.3563,C -0.0773,E1 12.3736,E2 366.5616} C_DIS
LIN {X 10.8186,Y 134.0856,Z 164,A 85.5222,B 12.3563,C -0.0801,E1 12.3687,E2 364.8123} C_DIS
LIN {X 7.2346,Y 134.3266,Z 164,A 86.7802,B 12.3563,C -0.0732,E1 12.3653,E2 363.5877} C_DIS
LIN {X 4.5793,Y 134.4442,Z 164,A 88.1782,B 12.3563,C -0.0801,E1 12.3613,E2 362.1582} C_DIS
LIN {X 0.5925,Y 134.5193,Z 164,A 89.7693,B 12.3563,C -0.0773,E1 12.3569,E2 360.5808} C_DIS
LIN {X -2.8191,Y 134.4922,Z 164,A 91.3043,B 12.3563,C -0.0792,E1 12.3526,E2 359.0367} C_DIS
LIN {X -6.4339,Y 134.3669,Z 164,A 92.6339,B 12.3563,C -0.0735,E1 12.3489,E2 357.7333} C_DIS
LIN {X -9.7231,Y 134.1686,Z 164,A 94.1536,B 12.3563,C -0.0762,E1 12.3447,E2 356.2003} C_DIS
LIN {X -13.2628,Y 133.8656,Z 164,A 95.769,B 12.3563,C -0.0782,E1 12.3401,E2 354.5734} C_DIS
LIN {X -17.6028,Y 133.3637,Z 164,A 97.5758,B 12.3563,C -0.0761,E1 12.3352,E2 352.7742} C_DIS
LIN {X -21.8813,Y 132.729,Z 164,A 99.3458,B 12.3563,C -0.0733,E1 12.3303,E2 351.0141} C_DIS
LIN {X -24.5529,Y 132.2625,Z 164,A 101.0615,B 12.3562,C -0.0868,E1 12.3254,E2 349.2315} C_DIS
LIN {X -28.8611,Y 131.3886,Z 164,A 102.4414,B 12.3562,C -0.073,E1 12.3218,E2 347.9124} C_DIS
LIN {X -32.9106,Y 130.4324,Z 164,A 104.1815,B 12.3562,C -0.0709,E1 12.3171,E2 346.1774} C_DIS
LIN {X -38.6091,Y 128.8626,Z 164,A 107.082,B 12.3562,C -0.0782,E1 12.3092,E2 343.2328} C_DIS
LIN {X -41.9754,Y 127.8046,Z 164,A 108.2871,B 12.3563,C -0.0694,E1 12.3061,E2 342.0648} C_DIS
LIN {X -44.9819,Y 126.7783,Z 164,A 109.6674,B 12.3563,C -0.0686,E1 12.3025,E2 340.6823} C_DIS
LIN {X -48.3736,Y 125.522,Z 164,A 111.184,B 12.3563,C -0.0663,E1 12.2985,E2 339.1698} C_DIS
LIN {X -51.735,Y 124.1738,Z 164,A 112.7801,B 12.3563,C -0.0658,E1 12.2944,E2 337.5686} C_DIS
LIN {X -56.0232,Y 122.2998,Z 164,A 114.5465,B 12.3563,C -0.0577,E1 12.2899,E2 335.8311} C_DIS
LIN {X -59.1099,Y 120.8381,Z 164,A 115.9969,B 12.3563,C -0.0557,E1 12.2863,E2 334.3825} C_DIS
LIN {X -61.9841,Y 119.39,Z 164,A 117.7706,B 12.3563,C -0.0635,E1 12.2818,E2 332.5618} C_DIS
LIN {X -66.5047,Y 116.9329,Z 164,A 119.8126,B 12.3563,C -0.0566,E1 12.2768,E2 330.5398} C_DIS
LIN {X -70.2231,Y 114.7383,Z 164,A 121.6832,B 12.3563,C -0.0545,E1 12.2723,E2 328.6672} C_DIS
LIN {X -73.8772,Y 112.4203,Z 164,A 123.5272,B 12.3563,C -0.0514,E1 12.268,E2 326.8249} C_DIS
LIN {X -77.5318,Y 109.9317,Z 164,A 125.3974,B 12.3564,C -0.0478,E1 12.2637,E2 324.9582} C_DIS
LIN {X -80.944,Y 107.4441,Z 164,A 127.2364,B 12.3564,C -0.0455,E1 12.2596,E2 323.1162} C_DIS
LIN {X -84.3336,Y 104.8046,Z 164,A 129.0708,B 12.3564,C -0.0422,E1 12.2556,E2 321.2832} C_DIS
LIN {X -87.6974,Y 102.0065,Z 164,A 130.9597,B 12.3564,C -0.0391,E1 12.2516,E2 319.3932} C_DIS
LIN {X -90.9897,Y 99.0809,Z 164,A 132.8598,B 12.3564,C -0.0358,E1 12.2476,E2 317.4922} C_DIS
LIN {X -94.1406,Y 96.0921,Z 164,A 134.7082,B 12.3564,C -0.0319,E1 12.2439,E2 315.646} C_DIS
LIN {X -97.2725,Y 92.9205,Z 164,A 136.6144,B 12.3564,C -0.028,E1 12.2402,E2 313.741} C_DIS
LIN {X -100.2143,Y 89.7398,Z 164,A 138.4968,B 12.3564,C -0.0247,E1 12.2367,E2 311.8563} C_DIS
LIN {X -103.0456,Y 86.474,Z 164,A 140.3367,B 12.3564,C -0.0204,E1 12.2333,E2 310.0185} C_DIS
LIN {X -105.8459,Y 83.0229,Z 164,A 142.2467,B 12.3564,C -0.0164,E1 12.23,E2 308.1087} C_DIS
LIN {X -108.5427,Y 79.4649,Z 164,A 144.2016,B 12.3564,C -0.013,E1 12.2267,E2 306.1496} C_DIS
LIN {X -111.1482,Y 75.7786,Z 164,A 146.1553,B 12.3564,C -0.009,E1 12.2236,E2 304.1943} C_DIS
LIN {X -112.8576,Y 73.2073,Z 164,A 147.5013,B 12.3564,C -0.0064,E1 12.2216,E2 302.8462} C_DIS
LIN {X -115.9558,Y 68.1938,Z 164,A 150.3039,B 12.3564,C -0.0067,E1 12.2175,E2 300.0111} C_DIS
LIN {X -117.7925,Y 64.9692,Z 164,A 151.6331,B 12.3564,C 0.0033,E1 12.2157,E2 298.7143} C_DIS
LIN {X -119.8349,Y 61.1164,Z 164,A 153.1801,B 12.3564,C 0.0154,E1 12.2138,E2 297.2068} C_DIS
LIN {X -121.3494,Y 58.0511,Z 164,A 154.6915,B 12.3564,C 0.0181,E1 12.2119,E2 295.6905} C_DIS
LIN {X -122.5949,Y 55.3746,Z 164,A 156.2129,B 12.3564,C 0.0154,E1 12.2101,E2 294.1389} C_DIS
LIN {X -123.9394,Y 52.2961,Z 164,A 157.6296,B 12.3564,C 0.0197,E1 12.2086,E2 292.7256} C_DIS
LIN {X -125.0829,Y 49.5033,Z 164,A 159.0321,B 12.3564,C 0.0206,E1 12.2071,E2 291.3106} C_DIS
LIN {X -126.5223,Y 45.6918,Z 164,A 160.6377,B 12.3564,C 0.0284,E1 12.2056,E2 289.7226} C_DIS
LIN {X -127.6859,Y 42.3318,Z 164,A 162.1712,B 12.3564,C 0.0323,E1 12.2042,E2 288.1886} C_DIS
LIN {X -128.8681,Y 38.592,Z 164,A 164.0193,B 12.3564,C 0.033,E1 12.2027,E2 286.3211} C_DIS
LIN {X -129.7063,Y 35.669,Z 164,A 165.2019,B 12.3564,C 0.0393,E1 12.2018,E2 285.1536} C_DIS
LIN {X -130.5097,Y 32.6061,Z 164,A 166.6599,B 12.3564,C 0.0407,E1 12.2008,E2 283.684} C_DIS
LIN {X -131.3044,Y 29.2467,Z 164,A 168.1469,B 12.3564,C 0.0446,E1 12.1999,E2 282.1968} C_DIS
LIN {X -132.0698,Y 25.5609,Z 164,A 169.6624,B 12.3564,C 0.0513,E1 12.199,E2 280.6938} C_DIS
LIN {X -133.0527,Y 19.8313,Z 164,A 172.3046,B 12.3564,C 0.0548,E1 12.1978,E2 278.0344} C_DIS
LIN {X -133.5567,Y 16.0734,Z 164,A 173.8004,B 12.3564,C 0.0622,E1 12.1973,E2 276.5549} C_DIS
LIN {X -133.9529,Y 12.354,Z 164,A 175.5198,B 12.3564,C 0.0641,E1 12.1969,E2 274.822} C_DIS
LIN {X -134.2905,Y 7.8725,Z 164,A 177.4519,B 12.3564,C 0.0693,E1 12.1965,E2 272.8899} C_DIS
LIN {X -134.4617,Y 3.9837,Z 164,A 179.0516,B 12.3563,C 0.0756,E1 12.1963,E2 271.299} C_DIS
LIN {X -134.5218,Y 0.1142,Z 164,A -179.3023,B 12.3563,C 0.0805,E1 12.1963,E2 269.6551} C_DIS
LIN {X -134.4814,Y -3.2761,Z 164,A -177.7792,B 12.3563,C 0.083,E1 12.1963,E2 268.1239} C_DIS
LIN {X -134.3325,Y -7.1178,Z 164,A -176.0632,B 12.3562,C 0.086,E1 12.1966,E2 266.4001} C_DIS
LIN {X -134.0418,Y -11.3369,Z 164,A -174.3971,B 12.3562,C 0.0944,E1 12.197,E2 264.7524} C_DIS
LIN {X -133.7167,Y -14.6853,Z 164,A -172.9006,B 12.3562,C 0.0971,E1 12.1974,E2 263.2496} C_DIS
LIN {X -133.2151,Y -18.6964,Z 164,A -171.1,B 12.3561,C 0.1004,E1 12.1981,E2 261.4412} C_DIS
LIN {X -132.5373,Y -23.0223,Z 164,A -169.3473,B 12.3561,C 0.1084,E1 12.1988,E2 259.7041} C_DIS
LIN {X -131.5855,Y -27.9489,Z 164,A -167.0571,B 12.3561,C 0.111,E1 12.2001,E2 257.3975} C_DIS
LIN {X -130.8341,Y -31.2757,Z 164,A -165.768,B 12.3559,C 0.1189,E1 12.2009,E2 256.1296} C_DIS
LIN {X -129.1983,Y -37.4645,Z 164,A -163.0117,B 12.3559,C 0.126,E1 12.2029,E2 253.3723} C_DIS
LIN {X -128.3766,Y -40.1959,Z 164,A -161.5724,B 12.3559,C 0.1242,E1 12.2041,E2 251.907} C_DIS
LIN {X -127.2169,Y -43.7224,Z 164,A -160.0306,B 12.3559,C 0.1295,E1 12.2055,E2 250.3713} C_DIS
LIN {X -126.0244,Y -47.0479,Z 164,A -158.6363,B 12.3558,C 0.1362,E1 12.2068,E2 248.9918} C_DIS
LIN {X -124.9545,Y -49.8223,Z 164,A -157.2014,B 12.3558,C 0.1357,E1 12.2083,E2 247.5373} C_DIS
LIN {X -123.4929,Y -53.3397,Z 164,A -155.5771,B 12.3558,C 0.14,E1 12.2101,E2 245.9142} C_DIS
LIN {X -121.9563,Y -56.7662,Z 164,A -153.8817,B 12.3557,C 0.142,E1 12.212,E2 244.2083} C_DIS
LIN {X -119.9065,Y -60.9758,Z 164,A -152.0106,B 12.3556,C 0.1501,E1 12.2143,E2 242.3538} C_DIS
LIN {X -118.3034,Y -64.036,Z 164,A -150.371,B 12.3556,C 0.1499,E1 12.2165,E2 240.6948} C_DIS
LIN {X -116.0566,Y -68.0222,Z 164,A -148.4446,B 12.3556,C 0.1553,E1 12.2192,E2 238.7726} C_DIS
LIN {X -114.0916,Y -71.2693,Z 164,A -146.8861,B 12.3555,C 0.1607,E1 12.2215,E2 237.2224} C_DIS
LIN {X -111.9312,Y -74.6161,Z 164,A -145.1747,B 12.3555,C 0.1644,E1 12.2241,E2 235.5102} C_DIS
LIN {X -109.6687,Y -77.9043,Z 164,A -143.3309,B 12.3555,C 0.165,E1 12.2271,E2 233.6498} C_DIS
LIN {X -106.992,Y -81.5409,Z 164,A -141.3988,B 12.3554,C 0.1692,E1 12.2303,E2 231.7178} C_DIS
LIN {X -104.0797,Y -85.2266,Z 164,A -139.4829,B 12.3553,C 0.1757,E1 12.2336,E2 229.8135} C_DIS
LIN {X -101.6182,Y -88.1478,Z 164,A -137.9492,B 12.3552,C 0.1815,E1 12.2364,E2 228.2921} C_DIS
LIN {X -99.3381,Y -90.7097,Z 164,A -136.2854,B 12.3552,C 0.1797,E1 12.2396,E2 226.6041} C_DIS
LIN {X -96.3539,Y -93.8736,Z 164,A -134.3832,B 12.3552,C 0.1823,E1 12.2432,E2 224.6967} C_DIS
LIN {X -93.3087,Y -96.9008,Z 164,A -132.5991,B 12.3552,C 0.187,E1 12.2468,E2 222.9188} C_DIS
LIN {X -90.1829,Y -99.8162,Z 164,A -130.8449,B 12.355,C 0.1921,E1 12.2504,E2 221.1735} C_DIS
LIN {X -87.4192,Y -102.2456,Z 164,A -129.1767,B 12.355,C 0.1925,E1 12.2539,E2 219.4934} C_DIS
LIN {X -83.8583,Y -105.1853,Z 164,A -127.1994,B 12.355,C 0.1957,E1 12.2582,E2 217.5155} C_DIS
LIN {X -80.3211,Y -107.9104,Z 164,A -125.2721,B 12.355,C 0.1983,E1 12.2625,E2 215.5856} C_DIS
LIN {X -76.6511,Y -110.5478,Z 164,A -123.3246,B 12.3549,C 0.2008,E1 12.267,E2 213.6357} C_DIS
LIN {X -72.6713,Y -113.2036,Z 164,A -120.7246,B 12.3551,C 0.1898,E1 12.2732,E2 210.9663} C_DIS
LIN {X -68.3374,Y -115.8711,Z 164,A -119.0895,B 12.3548,C 0.2062,E1 12.277,E2 209.3977} C_DIS
LIN {X -64.5322,Y -118.0329,Z 164,A -117.2165,B 12.3548,C 0.2085,E1 12.2816,E2 207.5239} C_DIS
LIN {X -61.6172,Y -119.5799,Z 164,A -115.9778,B 12.3547,C 0.2144,E1 12.2846,E2 206.306} C_DIS
LIN {X -58.2664,Y -121.2466,Z 164,A -114.2955,B 12.3547,C 0.2141,E1 12.2888,E2 204.6128} C_DIS
LIN {X -55.1198,Y -122.7089,Z 164,A -112.9185,B 12.3546,C 0.2183,E1 12.2923,E2 203.2483} C_DIS
LIN {X -52.6357,Y -123.7973,Z 164,A -111.5015,B 12.3546,C 0.2129,E1 12.296,E2 201.7989} C_DIS
LIN {X -49.0456,Y -125.2608,Z 164,A -109.9865,B 12.3546,C 0.2179,E1 12.2999,E2 200.3007} C_DIS
LIN {X -45.9238,Y -126.4387,Z 164,A -108.4862,B 12.3546,C 0.2172,E1 12.3038,E2 198.7905} C_DIS
LIN {X -42.5646,Y -127.6084,Z 164,A -107.182,B 12.3545,C 0.2238,E1 12.3072,E2 197.5123} C_DIS
LIN {X -40.2183,Y -128.3694,Z 164,A -105.8491,B 12.3546,C 0.2174,E1 12.3109,E2 196.1444} C_DIS
LIN {X -36.9447,Y -129.3495,Z 164,A -104.4602,B 12.3546,C 0.2201,E1 12.3146,E2 194.7635} C_DIS
LIN {X -33.2365,Y -130.3497,Z 164,A -103.0226,B 12.3545,C 0.2262,E1 12.3184,E2 193.3502} C_DIS
LIN {X -30.1894,Y -131.0891,Z 164,A -101.5755,B 12.3545,C 0.2241,E1 12.3224,E2 191.8889} C_DIS
LIN {X -26.7679,Y -131.8301,Z 164,A -100.13,B 12.3545,C 0.226,E1 12.3263,E2 190.4488} C_DIS
LIN {X -24.1441,Y -132.3366,Z 164,A -99.0627,B 12.3545,C 0.2283,E1 12.3292,E2 189.39} C_DIS
LIN {X -21.2794,Y -132.8284,Z 164,A -97.6062,B 12.3545,C 0.223,E1 12.3333,E2 187.906} C_DIS
LIN {X -17.7165,Y -133.3488,Z 164,A -96.1221,B 12.3545,C 0.2247,E1 12.3374,E2 186.4275} C_DIS
LIN {X -14.1671,Y -133.7725,Z 164,A -94.6538,B 12.3545,C 0.2264,E1 12.3414,E2 184.9654} C_DIS
LIN {X -10.4044,Y -134.1189,Z 164,A -93.0506,B 12.3545,C 0.2268,E1 12.3459,E2 183.3624} C_DIS
LIN {X -7.6022,Y -134.3071,Z 164,A -91.6927,B 12.3545,C 0.2226,E1 12.3497,E2 181.9839} C_DIS
LIN {X -3.739,Y -134.4685,Z 164,A -90.1539,B 12.3545,C 0.2254,E1 12.354,E2 180.4578} C_DIS
LIN {X 0.0182,Y -134.5225,Z 164,A -88.4406,B 12.3545,C 0.2222,E1 12.3588,E2 178.7297} C_DIS
LIN {X 0.0182,Y -134.5225,Z 164,A -88.4406,B 12.3545,C 0.2222,E1 12.3588,E2 178.7297} C_DIS
Enddeposition()
LIN {X 0.9829,Y -135.4364,Z 164,A -88.4961,B 12.2768,C 0.2465,E1 12.2811,E2 178.9014} C_DIS
Startdeposition()
$VEL.CP = VEL_PRINT
LIN {X -1.4998,Y -135.434,Z 164,A -89.7661,B 12.2768,C 0.2525,E1 12.2775,E2 180.1994} C_DIS
LIN {X -5.4581,Y -135.3302,Z 164,A -91.4997,B 12.2767,C 0.2541,E1 12.2726,E2 181.9409} C_DIS
LIN {X -9.0934,Y -135.1367,Z 164,A -92.9871,B 12.2767,C 0.2527,E1 12.2685,E2 183.4225} C_DIS
LIN {X -12.1037,Y -134.9,Z 164,A -94.2687,B 12.2767,C 0.2527,E1 12.2649,E2 184.7051} C_DIS
LIN {X -15.0661,Y -134.6007,Z 164,A -95.4853,B 12.2767,C 0.2513,E1 12.2616,E2 185.9168} C_DIS
LIN {X -17.6959,Y -134.279,Z 164,A -96.6862,B 12.2767,C 0.2531,E1 12.2582,E2 187.1279} C_DIS
LIN {X -21.4388,Y -133.7344,Z 164,A -98.2605,B 12.2767,C 0.252,E1 12.2539,E2 188.6997} C_DIS
LIN {X -24.6455,Y -133.1811,Z 164,A -99.6404,B 12.2767,C 0.2515,E1 12.2501,E2 190.0803} C_DIS
LIN {X -27.3214,Y -132.656,Z 164,A -100.8404,B 12.2767,C 0.2522,E1 12.2468,E2 191.2863} C_DIS
LIN {X -30.6452,Y -131.9283,Z 164,A -102.2621,B 12.2767,C 0.251,E1 12.2429,E2 192.7061} C_DIS
LIN {X -34.0402,Y -131.0945,Z 164,A -103.7217,B 12.2767,C 0.2496,E1 12.239,E2 194.1637} C_DIS
LIN {X -37.2681,Y -130.214,Z 164,A -105.1485,B 12.2767,C 0.249,E1 12.2351,E2 195.5922} C_DIS
LIN {X -39.9463,Y -129.4153,Z 164,A -106.3758,B 12.2767,C 0.2492,E1 12.2318,E2 196.8251} C_DIS
LIN {X -43.5784,Y -128.2401,Z 164,A -107.9588,B 12.2768,C 0.2472,E1 12.2276,E2 198.4044} C_DIS
LIN {X -46.6551,Y -127.1527,Z 164,A -109.3357,B 12.2768,C 0.2459,E1 12.224,E2 199.781} C_DIS
LIN {X -49.4345,Y -126.0963,Z 164,A -110.647,B 12.2768,C 0.246,E1 12.2206,E2 201.0989} C_DIS
LIN {X -52.9068,Y -124.681,Z 164,A -112.2052,B 12.2768,C 0.2437,E1 12.2166,E2 202.6537} C_DIS
LIN {X -56.0075,Y -123.3193,Z 164,A -113.6365,B 12.2769,C 0.2421,E1 12.2129,E2 204.0848} C_DIS
LIN {X -59.1533,Y -121.8421,Z 164,A -115.1245,B 12.2769,C 0.2409,E1 12.2092,E2 205.5749} C_DIS
LIN {X -62.2079,Y -120.3112,Z 164,A -116.5787,B 12.2769,C 0.2393,E1 12.2055,E2 207.0301} C_DIS
LIN {X -65.2347,Y -118.6973,Z 164,A -118.029,B 12.277,C 0.2374,E1 12.202,E2 208.4802} C_DIS
LIN {X -68.2304,Y -117.0009,Z 164,A -119.5049,B 12.277,C 0.2359,E1 12.1984,E2 209.9583} C_DIS
LIN {X -71.1917,Y -115.223,Z 164,A -120.9757,B 12.277,C 0.2341,E1 12.1949,E2 211.4301} C_DIS
LIN {X -74.2789,Y -113.2569,Z 164,A -122.6472,B 12.277,C 0.2348,E1 12.1909,E2 213.1164} C_DIS
LIN {X -78.0054,Y -110.723,Z 164,A -124.5365,B 12.2771,C 0.2314,E1 12.1866,E2 215.0032} C_DIS
LIN {X -81.2083,Y -108.3965,Z 164,A -126.2396,B 12.2771,C 0.2293,E1 12.1828,E2 216.7094} C_DIS
LIN {X -84.6592,Y -105.7232,Z 164,A -128.0027,B 12.2773,C 0.2241,E1 12.1789,E2 218.4617} C_DIS
LIN {X -87.3611,Y -103.5017,Z 164,A -129.4977,B 12.2773,C 0.2218,E1 12.1757,E2 219.958} C_DIS
LIN {X -90.3392,Y -100.9121,Z 164,A -131.222,B 12.2773,C 0.22,E1 12.1721,E2 221.6883} C_DIS
LIN {X -93.3429,Y -98.1408,Z 164,A -133.0378,B 12.2773,C 0.2187,E1 12.1684,E2 223.5141} C_DIS
LIN {X -96.5855,Y -94.9509,Z 164,A -134.956,B 12.2774,C 0.2147,E1 12.1646,E2 225.4307} C_DIS
LIN {X -99.4176,Y -91.9823,Z 164,A -136.6893,B 12.2774,C 0.2111,E1 12.1613,E2 227.163} C_DIS
LIN {X -102.3394,Y -88.7201,Z 164,A -138.4806,B 12.2776,C 0.2057,E1 12.158,E2 228.9458} C_DIS
LIN {X -104.9553,Y -85.6085,Z 164,A -140.2584,B 12.2776,C 0.2033,E1 12.1548,E2 230.7297} C_DIS
LIN {X -107.3183,Y -82.6279,Z 164,A -141.9183,B 12.2776,C 0.2008,E1 12.1519,E2 232.395} C_DIS
LIN {X -109.9169,Y -79.1383,Z 164,A -143.8191,B 12.2776,C 0.198,E1 12.1488,E2 234.3021} C_DIS
LIN {X -112.4055,Y -75.562,Z 164,A -145.6839,B 12.2778,C 0.1941,E1 12.1458,E2 236.1683} C_DIS
LIN {X -114.746,Y -71.9578,Z 164,A -147.4516,B 12.2778,C 0.1885,E1 12.1432,E2 237.9286} C_DIS
LIN {X -116.9821,Y -68.2624,Z 164,A -149.2389,B 12.2779,C 0.1831,E1 12.1406,E2 239.7098} C_DIS
LIN {X -118.6793,Y -65.2671,Z 164,A -150.7135,B 12.2779,C 0.1798,E1 12.1386,E2 241.1856} C_DIS
LIN {X -120.3112,Y -62.2079,Z 164,A -152.1912,B 12.278,C 0.1763,E1 12.1367,E2 242.6635} C_DIS
LIN {X -121.8096,Y -59.2192,Z 164,A -153.6198,B 12.278,C 0.1729,E1 12.1349,E2 244.0928} C_DIS
LIN {X -123.2588,Y -56.1405,Z 164,A -155.075,B 12.2781,C 0.1695,E1 12.1332,E2 245.5487} C_DIS
LIN {X -124.6378,Y -53.0091,Z 164,A -156.5305,B 12.2781,C 0.1658,E1 12.1316,E2 247.004} C_DIS
LIN {X -125.799,Y -50.1871,Z 164,A -157.8642,B 12.2781,C 0.1633,E1 12.1302,E2 248.3418} C_DIS
LIN {X -127.1283,Y -46.7227,Z 164,A -159.4265,B 12.2783,C 0.1589,E1 12.1287,E2 249.9019} C_DIS
LIN {X -128.0938,Y -44.0005,Z 164,A -160.6798,B 12.2783,C 0.1562,E1 12.1275,E2 251.1579} C_DIS
LIN {X -129.2686,Y -40.4258,Z 164,A -162.2694,B 12.2783,C 0.1518,E1 12.1262,E2 252.7459} C_DIS
LIN {X -130.1941,Y -37.3361,Z 164,A -163.6416,B 12.2783,C 0.1481,E1 12.1251,E2 254.1178} C_DIS
LIN {X -131.0591,Y -34.1762,Z 164,A -165.0504,B 12.2784,C 0.1447,E1 12.1241,E2 255.528} C_DIS
LIN {X -131.8177,Y -31.1198,Z 164,A -166.3941,B 12.2784,C 0.1412,E1 12.1232,E2 256.8718} C_DIS
LIN {X -132.5451,Y -27.862,Z 164,A -167.8236,B 12.2785,C 0.1375,E1 12.1223,E2 258.302} C_DIS
LIN {X -133.1682,Y -24.7132,Z 164,A -169.1932,B 12.2785,C 0.1339,E1 12.1216,E2 259.6717} C_DIS
LIN {X -133.7127,Y -21.5737,Z 164,A -170.5579,B 12.2785,C 0.1303,E1 12.121,E2 261.0372} C_DIS
LIN {X -134.1376,Y -18.7423,Z 164,A -171.792,B 12.2786,C 0.1273,E1 12.1205,E2 262.2728} C_DIS
LIN {X -134.5668,Y -15.3694,Z 164,A -173.2374,B 12.2786,C 0.1233,E1 12.12,E2 263.7175} C_DIS
LIN {X -134.888,Y -12.2366,Z 164,A -174.5643,B 12.2786,C 0.1192,E1 12.1197,E2 265.0424} C_DIS
LIN {X -135.2173,Y -7.7844,Z 164,A -176.4814,B 12.2787,C 0.1143,E1 12.1193,E2 266.9609} C_DIS
LIN {X -135.3668,Y -4.5191,Z 164,A -177.8873,B 12.2787,C 0.1108,E1 12.1191,E2 268.3682} C_DIS
LIN {X -135.4359,Y -1.2077,Z 164,A -179.4169,B 12.2787,C 0.1095,E1 12.1191,E2 269.9117} C_DIS
LIN {X -135.4222,Y 2.2083,Z 164,A 179.2085,B 12.2788,C 0.1036,E1 12.1191,E2 271.2763} C_DIS
LIN {X -135.3278,Y 5.5192,Z 164,A 177.8083,B 12.2788,C 0.0995,E1 12.1192,E2 272.6747} C_DIS
LIN {X -135.1367,Y 9.0934,Z 164,A 176.2736,B 12.2788,C 0.0955,E1 12.1195,E2 274.2103} C_DIS
LIN {X -134.9,Y 12.1037,Z 164,A 174.9765,B 12.2789,C 0.0921,E1 12.1198,E2 275.5083} C_DIS
LIN {X -134.6368,Y 14.7305,Z 164,A 173.7912,B 12.2789,C 0.0904,E1 12.1201,E2 276.7006} C_DIS
LIN {X -134.1983,Y 18.3118,Z 164,A 172.2965,B 12.2789,C 0.0852,E1 12.1207,E2 278.1897} C_DIS
LIN {X -133.7344,Y 21.4388,Z 164,A 170.9461,B 12.2789,C 0.0815,E1 12.1212,E2 279.5402} C_DIS
LIN {X -133.2922,Y 24.0248,Z 164,A 169.7741,B 12.279,C 0.0797,E1 12.1218,E2 280.7183} C_DIS
LIN {X -132.5736,Y 27.7262,Z 164,A 168.203,B 12.279,C 0.0745,E1 12.1227,E2 282.2847} C_DIS
LIN {X -131.8743,Y 30.8813,Z 164,A 166.8098,B 12.279,C 0.0711,E1 12.1235,E2 283.6795} C_DIS
LIN {X -131.0945,Y 34.0402,Z 164,A 165.4145,B 12.279,C 0.0676,E1 12.1245,E2 285.0755} C_DIS
LIN {X -130.214,Y 37.2681,Z 164,A 163.9812,B 12.2791,C 0.0639,E1 12.1256,E2 286.5093} C_DIS
LIN {X -129.4102,Y 39.963,Z 164,A 162.7379,B 12.2791,C 0.0617,E1 12.1266,E2 287.7576} C_DIS
LIN {X -128.2401,Y 43.5784,Z 164,A 161.1461,B 12.2791,C 0.0568,E1 12.128,E2 289.3456} C_DIS
LIN {X -127.1527,Y 46.6551,Z 164,A 159.7474,B 12.2791,C 0.0533,E1 12.1293,E2 290.7449} C_DIS
LIN {X -125.9588,Y 49.7882,Z 164,A 158.3188,B 12.2791,C 0.0496,E1 12.1307,E2 292.173} C_DIS
LIN {X -124.681,Y 52.9068,Z 164,A 156.8665,B 12.2791,C 0.0463,E1 12.1323,E2 293.6268} C_DIS
LIN {X -123.3193,Y 56.0075,Z 164,A 155.4145,B 12.2791,C 0.0428,E1 12.134,E2 295.0794} C_DIS
LIN {X -121.8421,Y 59.1533,Z 164,A 153.9273,B 12.2792,C 0.0392,E1 12.1358,E2 296.567} C_DIS
LIN {X -120.3112,Y 62.2079,Z 164,A 152.464,B 12.2792,C 0.0358,E1 12.1376,E2 298.0306} C_DIS
LIN {X -118.2809,Y 65.9867,Z 164,A 150.6275,B 12.2792,C 0.0315,E1 12.1401,E2 299.8676} C_DIS
LIN {X -116.5641,Y 68.9741,Z 164,A 149.1528,B 12.2792,C 0.0281,E1 12.1421,E2 301.3427} C_DIS
LIN {X -114.7659,Y 71.9263,Z 164,A 147.6735,B 12.2792,C 0.0247,E1 12.1443,E2 302.8223} C_DIS
LIN {X -112.908,Y 74.8088,Z 164,A 146.0883,B 12.2792,C 0.0241,E1 12.1468,E2 304.4219} C_DIS
LIN {X -110.4284,Y 78.423,Z 164,A 144.3318,B 12.2792,C 0.0173,E1 12.1495,E2 306.1646} C_DIS
LIN {X -108.3965,Y 81.2083,Z 164,A 142.7955,B 12.2792,C 0.0156,E1 12.1521,E2 307.7085} C_DIS
LIN {X -105.7232,Y 84.6592,Z 164,A 140.9916,B 12.2792,C 0.0102,E1 12.1552,E2 309.5051} C_DIS
LIN {X -103.5017,Y 87.3611,Z 164,A 139.4933,B 12.2792,C 0.0072,E1 12.1579,E2 311.004} C_DIS
LIN {X -101.2087,Y 90.0077,Z 164,A 138.0168,B 12.2792,C 0.0037,E1 12.1606,E2 312.4782} C_DIS
LIN {X -98.666,Y 92.7873,Z 164,A 136.2845,B 12.2792,C 0.0034,E1 12.1639,E2 314.2254} C_DIS
LIN {X -95.7987,Y 95.7454,Z 164,A 134.6296,B 12.2792,C -0.0024,E1 12.1671,E2 315.8678} C_DIS
LIN {X -93.2884,Y 98.1929,Z 164,A 133.1332,B 12.2792,C -0.0052,E1 12.1701,E2 317.3642} C_DIS
LIN {X -90.7572,Y 100.5369,Z 164,A 131.5955,B 12.2792,C -0.0064,E1 12.1733,E2 318.9097} C_DIS
LIN {X -87.4187,Y 103.4531,Z 164,A 129.7745,B 12.2792,C -0.0114,E1 12.1772,E2 320.7222} C_DIS
LIN {X -84.6886,Y 105.6998,Z 164,A 128.2669,B 12.2792,C -0.014,E1 12.1804,E2 322.2296} C_DIS
LIN {X -81.9047,Y 107.8712,Z 164,A 126.6385,B 12.2792,C -0.0136,E1 12.1841,E2 323.8725} C_DIS
LIN {X -78.2655,Y 110.5395,Z 164,A 124.726,B 12.2792,C -0.0169,E1 12.1884,E2 325.7835} C_DIS
LIN {X -74.84,Y 112.8875,Z 164,A 123.0709,B 12.2792,C -0.0223,E1 12.1922,E2 327.4248} C_DIS
LIN {X -71.9578,Y 114.746,Z 164,A 121.5024,B 12.2792,C -0.0219,E1 12.1959,E2 329.0059} C_DIS
LIN {X -68.2624,Y 116.9821,Z 164,A 119.7729,B 12.2792,C -0.0271,E1 12.2,E2 330.7219} C_DIS
LIN {X -65.2671,Y 118.6793,Z 164,A 118.3047,B 12.2792,C -0.029,E1 12.2036,E2 332.1903} C_DIS
LIN {X -62.2079,Y 120.3112,Z 164,A 116.834,B 12.2792,C -0.031,E1 12.2072,E2 333.66} C_DIS
LIN {X -59.567,Y 121.638,Z 164,A 115.5453,B 12.2792,C -0.0318,E1 12.2105,E2 334.9521} C_DIS
LIN {X -56.1405,Y 123.2588,Z 164,A 113.9658,B 12.2792,C -0.0345,E1 12.2145,E2 336.5274} C_DIS
LIN {X -52.9738,Y 124.653,Z 164,A 112.497,B 12.2792,C -0.0362,E1 12.2182,E2 337.9956} C_DIS
LIN {X -49.9703,Y 125.8864,Z 164,A 111.1292,B 12.2792,C -0.0379,E1 12.2218,E2 339.3615} C_DIS
LIN {X -46.7227,Y 127.1283,Z 164,A 109.6424,B 12.2792,C -0.0391,E1 12.2257,E2 340.8491} C_DIS
LIN {X -43.6461,Y 128.2166,Z 164,A 108.2602,B 12.2792,C -0.0405,E1 12.2293,E2 342.2304} C_DIS
LIN {X -40.4258,Y 129.2686,Z 164,A 106.8207,B 12.2792,C -0.0418,E1 12.2331,E2 343.6695} C_DIS
LIN {X -37.3361,Y 130.1941,Z 164,A 105.453,B 12.2792,C -0.0429,E1 12.2368,E2 345.0366} C_DIS
LIN {X -34.2178,Y 131.048,Z 164,A 104.0843,B 12.2792,C -0.044,E1 12.2405,E2 346.4044} C_DIS
LIN {X -31.3931,Y 131.7518,Z 164,A 102.811,B 12.2792,C -0.044,E1 12.2439,E2 347.6817} C_DIS
LIN {X -27.862,Y 132.5451,Z 164,A 101.3144,B 12.2792,C -0.0458,E1 12.248,E2 349.1732} C_DIS
LIN {X -24.7132,Y 133.1682,Z 164,A 99.9671,B 12.2792,C -0.0469,E1 12.2517,E2 350.5184} C_DIS
LIN {X -21.5737,Y 133.7127,Z 164,A 98.6066,B 12.2792,C -0.0474,E1 12.2555,E2 351.8795} C_DIS
LIN {X -18.3789,Y 134.1895,Z 164,A 97.2404,B 12.2792,C -0.048,E1 12.2592,E2 353.2449} C_DIS
LIN {X -15.333,Y 134.5712,Z 164,A 95.9552,B 12.2792,C -0.0489,E1 12.2628,E2 354.5276} C_DIS
LIN {X -12.5192,Y 134.8609,Z 164,A 94.7285,B 12.2792,C -0.0486,E1 12.2662,E2 355.7573} C_DIS
LIN {X -9.0934,Y 135.1367,Z 164,A 93.2932,B 12.2792,C -0.0494,E1 12.2702,E2 357.1896} C_DIS
LIN {X -6.038,Y 135.3076,Z 164,A 91.9996,B 12.2792,C -0.0497,E1 12.2738,E2 358.4824} C_DIS
LIN {X -3.0714,Y 135.4071,Z 164,A 90.7461,B 12.2792,C -0.05,E1 12.2773,E2 359.735} C_DIS
LIN {X 0.8331,Y 135.4376,Z 164,A 89.0458,B 12.2792,C -0.0489,E1 12.2821,E2 361.4403} C_DIS
LIN {X 4.5191,Y 135.3668,Z 164,A 87.5315,B 12.2792,C -0.05,E1 12.2863,E2 362.9486} C_DIS
LIN {X 7.4972,Y 135.2342,Z 164,A 86.2669,B 12.2792,C -0.0498,E1 12.2898,E2 364.2131} C_DIS
LIN {X 10.563,Y 135.0294,Z 164,A 84.9695,B 12.2792,C -0.0497,E1 12.2934,E2 365.5097} C_DIS
LIN {X 13.1861,Y 134.7968,Z 164,A 83.8618,B 12.2792,C -0.0497,E1 12.2965,E2 366.6162} C_DIS
LIN {X 16.4083,Y 134.4429,Z 164,A 82.4507,B 12.2792,C -0.0482,E1 12.3004,E2 368.0316} C_DIS
LIN {X 19.8736,Y 133.9759,Z 164,A 80.9996,B 12.2792,C -0.0484,E1 12.3044,E2 369.4788} C_DIS
LIN {X 23.0745,Y 133.4622,Z 164,A 79.6288,B 12.2792,C -0.0478,E1 12.3082,E2 370.8493} C_DIS
LIN {X 27.5463,Y 132.6102,Z 164,A 77.6905,B 12.2792,C -0.0465,E1 12.3135,E2 372.7886} C_DIS
LIN {X 30.8813,Y 131.8743,Z 164,A 76.2644,B 12.2792,C -0.0462,E1 12.3174,E2 374.2121} C_DIS
LIN {X 33.5333,Y 131.2231,Z 164,A 75.0699,B 12.2792,C -0.0444,E1 12.3206,E2 375.411} C_DIS
LIN {X 37.2681,Y 130.214,Z 164,A 73.4728,B 12.2792,C -0.0442,E1 12.3249,E2 377.0033} C_DIS
LIN {X 40.4258,Y 129.2686,Z 164,A 72.0812,B 12.2792,C -0.0432,E1 12.3286,E2 378.3943} C_DIS
LIN {X 43.5784,Y 128.2401,Z 164,A 70.6814,B 12.2792,C -0.042,E1 12.3323,E2 379.7937} C_DIS
LIN {X 46.2644,Y 127.2935,Z 164,A 69.4429,B 12.2792,C -0.04,E1 12.3356,E2 381.036} C_DIS
LIN {X 49.7882,Y 125.9588,Z 164,A 67.8893,B 12.2792,C -0.0395,E1 12.3396,E2 382.5847} C_DIS
LIN {X 52.9068,Y 124.681,Z 164,A 66.4715,B 12.2792,C -0.0382,E1 12.3433,E2 384.0016} C_DIS
LIN {X 55.924,Y 123.3566,Z 164,A 65.0754,B 12.2792,C -0.0365,E1 12.3468,E2 385.3979} C_DIS
LIN {X 59.1533,Y 121.8421,Z 164,A 63.5784,B 12.2792,C -0.035,E1 12.3506,E2 386.8936} C_DIS
LIN {X 62.2079,Y 120.3112,Z 164,A 62.1393,B 12.2792,C -0.0333,E1 12.3542,E2 388.332} C_DIS
LIN {X 66.7044,Y 117.8775,Z 164,A 59.9833,B 12.2792,C -0.0305,E1 12.3595,E2 390.4875} C_DIS
LIN {X 69.7156,Y 116.1221,Z 164,A 58.4135,B 12.2792,C -0.0258,E1 12.3633,E2 392.069} C_DIS
LIN {X 73.3881,Y 113.8367,Z 164,A 56.6033,B 12.2792,C -0.0235,E1 12.3675,E2 393.8772} C_DIS
LIN {X 76.998,Y 111.4267,Z 164,A 54.8758,B 12.2792,C -0.0235,E1 12.3715,E2 395.592} C_DIS
LIN {X 79.8366,Y 109.4108,Z 164,A 53.3422,B 12.2792,C -0.0194,E1 12.375,E2 397.1333} C_DIS
LIN {X 83.2883,Y 106.8065,Z 164,A 51.5961,B 12.2792,C -0.0186,E1 12.3788,E2 398.8699} C_DIS
LIN {X 86.0169,Y 104.6215,Z 164,A 50.1279,B 12.2792,C -0.0162,E1 12.382,E2 400.3373} C_DIS
LIN {X 88.7201,Y 102.3394,Z 164,A 48.5435,B 12.2792,C -0.0109,E1 12.3854,E2 401.9329} C_DIS
LIN {X 91.9545,Y 99.4432,Z 164,A 46.8167,B 12.2792,C -0.0104,E1 12.389,E2 403.6471} C_DIS
LIN {X 94.9041,Y 96.6315,Z 164,A 45.0626,B 12.2792,C -0.0061,E1 12.3925,E2 405.4056} C_DIS
LIN {X 97.8645,Y 93.632,Z 164,A 43.2627,B 12.2792,C -0.002,E1 12.396,E2 407.2083} C_DIS
LIN {X 100.5993,Y 90.6884,Z 164,A 41.6696,B 12.2792,C -0.0013,E1 12.399,E2 408.7893} C_DIS
LIN {X 103.0737,Y 87.865,Z 164,A 39.986,B 12.2792,C 0.0048,E1 12.4021,E2 410.4854} C_DIS
LIN {X 105.6998,Y 84.6886,Z 164,A 38.3584,B 12.2792,C 0.0055,E1 12.4049,E2 412.0999} C_DIS
LIN {X 107.8485,Y 81.9347,Z 164,A 36.7743,B 12.2792,C 0.0119,E1 12.4076,E2 413.6978} C_DIS
LIN {X 110.4066,Y 78.4535,Z 164,A 35.0822,B 12.2792,C 0.0124,E1 12.4104,E2 415.3746} C_DIS
LIN {X 112.4055,Y 75.562,Z 164,A 33.6152,B 12.2792,C 0.0154,E1 12.4127,E2 416.84} C_DIS
LIN {X 114.4356,Y 72.4496,Z 164,A 31.9616,B 12.2792,C 0.0215,E1 12.4152,E2 418.5046} C_DIS
LIN {X 116.545,Y 69.006,Z 164,A 30.3705,B 12.2792,C 0.0225,E1 12.4175,E2 420.0826} C_DIS
LIN {X 118.2809,Y 65.9867,Z 164,A 28.914,B 12.2792,C 0.0257,E1 12.4195,E2 421.5382} C_DIS
LIN {X 120.1216,Y 62.5689,Z 164,A 27.2978,B 12.2792,C 0.0292,E1 12.4216,E2 423.1523} C_DIS
LIN {X 121.8096,Y 59.2192,Z 164,A 25.7222,B 12.2792,C 0.033,E1 12.4236,E2 424.7278} C_DIS
LIN {X 123.164,Y 56.3456,Z 164,A 24.3991,B 12.2792,C 0.036,E1 12.4251,E2 426.0494} C_DIS
LIN {X 124.653,Y 52.9738,Z 164,A 22.8541,B 12.2792,C 0.0398,E1 12.4268,E2 427.5941} C_DIS
LIN {X 125.9055,Y 49.9228,Z 164,A 21.475,B 12.2792,C 0.0431,E1 12.4283,E2 428.9723} C_DIS
LIN {X 127.1283,Y 46.7227,Z 164,A 20.0451,B 12.2792,C 0.0465,E1 12.4297,E2 430.4011} C_DIS
LIN {X 128.0829,Y 44.0319,Z 164,A 18.8178,B 12.2792,C 0.0504,E1 12.4308,E2 431.6318} C_DIS
LIN {X 129.2686,Y 40.4258,Z 164,A 17.2676,B 12.2792,C 0.0533,E1 12.4321,E2 433.1767} C_DIS
LIN {X 130.1941,Y 37.3361,Z 164,A 15.9209,B 12.2792,C 0.0566,E1 12.4332,E2 434.5224} C_DIS
LIN {X 130.9351,Y 34.641,Z 164,A 14.7558,B 12.2792,C 0.0595,E1 12.434,E2 435.6865} C_DIS
LIN {X 131.7257,Y 31.5014,Z 164,A 13.404,B 12.2792,C 0.0629,E1 12.4349,E2 437.0374} C_DIS
LIN {X 132.4634,Y 28.2405,Z 164,A 11.994,B 12.2791,C 0.0668,E1 12.4358,E2 438.4483} C_DIS
LIN {X 133.1011,Y 25.0638,Z 164,A 10.6545,B 12.2791,C 0.0699,E1 12.4365,E2 439.7853} C_DIS
LIN {X 133.6351,Y 22.0387,Z 164,A 9.3228,B 12.2791,C 0.0746,E1 12.4371,E2 441.1223} C_DIS
LIN {X 134.1895,Y 18.3789,Z 164,A 7.8285,B 12.2791,C 0.0771,E1 12.4377,E2 442.6094} C_DIS
LIN {X 134.5712,Y 15.333,Z 164,A 6.5511,B 12.2791,C 0.0803,E1 12.4381,E2 443.8856} C_DIS
LIN {X 134.8244,Y 12.8987,Z 164,A 5.5157,B 12.279,C 0.0833,E1 12.4384,E2 444.922} C_DIS
LIN {X 135.0923,Y 9.7009,Z 164,A 4.1304,B 12.279,C 0.0881,E1 12.4387,E2 446.3121} C_DIS
LIN {X 135.3076,Y 6.038,Z 164,A 2.6583,B 12.279,C 0.0904,E1 12.4389,E2 447.7761} C_DIS
LIN {X 135.4071,Y 3.0714,Z 164,A 1.421,B 12.279,C 0.0935,E1 12.439,E2 449.0125} C_DIS
LIN {X 135.4421,Y 0,Z 164,A 0.1212,B 12.2789,C 0.0974,E1 12.439,E2 450.3138} C_DIS
LIN {X 135.3668,Y -4.5191,Z 164,A -1.7539,B 12.2789,C 0.102,E1 12.439,E2 452.1864} C_DIS
LIN {X 135.2342,Y -7.4972,Z 164,A -3.0034,B 12.2789,C 0.1054,E1 12.4388,E2 453.4359} C_DIS
LIN {X 135.0294,Y -10.563,Z 164,A -4.2885,B 12.2788,C 0.1088,E1 12.4385,E2 454.7207} C_DIS
LIN {X 134.765,Y -13.5177,Z 164,A -5.5092,B 12.2788,C 0.1115,E1 12.4382,E2 455.9385} C_DIS
LIN {X 134.4502,Y -16.3468,Z 164,A -6.7336,B 12.2788,C 0.1157,E1 12.4378,E2 457.1668} C_DIS
LIN {X 133.9759,Y -19.8736,Z 164,A -8.2117,B 12.2787,C 0.1193,E1 12.4372,E2 458.6433} C_DIS
LIN {X 133.4622,Y -23.0745,Z 164,A -9.5683,B 12.2787,C 0.1229,E1 12.4366,E2 459.9997} C_DIS
LIN {X 132.8803,Y -26.2188,Z 164,A -10.9069,B 12.2787,C 0.1265,E1 12.4359,E2 461.3382} C_DIS
LIN {X 132.2193,Y -29.371,Z 164,A -12.2551,B 12.2786,C 0.13,E1 12.4351,E2 462.6862} C_DIS
LIN {X 131.4782,Y -32.5284,Z 164,A -13.6124,B 12.2786,C 0.1336,E1 12.4342,E2 464.0433} C_DIS
LIN {X 130.6761,Y -35.6124,Z 164,A -14.9423,B 12.2786,C 0.137,E1 12.4333,E2 465.3726} C_DIS
LIN {X 129.8363,Y -38.5581,Z 164,A -16.227,B 12.2785,C 0.1404,E1 12.4323,E2 466.6574} C_DIS
LIN {X 128.7864,Y -41.935,Z 164,A -17.7102,B 12.2785,C 0.1443,E1 12.431,E2 468.1408} C_DIS
LIN {X 127.6947,Y -45.1518,Z 164,A -19.131,B 12.2784,C 0.1479,E1 12.4297,E2 469.5613} C_DIS
LIN {X 126.5662,Y -48.2232,Z 164,A -20.5007,B 12.2784,C 0.1514,E1 12.4284,E2 470.9309} C_DIS
LIN {X 125.3715,Y -51.2475,Z 164,A -21.8494,B 12.2784,C 0.1544,E1 12.427,E2 472.2779} C_DIS
LIN {X 124.0107,Y -54.4596,Z 164,A -23.3225,B 12.2783,C 0.1584,E1 12.4253,E2 473.7525} C_DIS
LIN {X 122.5763,Y -57.6166,Z 164,A -24.774,B 12.2783,C 0.162,E1 12.4236,E2 475.2039} C_DIS
LIN {X 121.0871,Y -60.6838,Z 164,A -26.2017,B 12.2782,C 0.1655,E1 12.4219,E2 476.6315} C_DIS
LIN {X 119.1291,Y -64.4424,Z 164,A -28.0717,B 12.2781,C 0.1725,E1 12.4194,E2 478.5131} C_DIS
LIN {X 117.0502,Y -68.1453,Z 164,A -29.7653,B 12.2781,C 0.1743,E1 12.4171,E2 480.1961} C_DIS
LIN {X 115.2033,Y -71.2233,Z 164,A -31.3795,B 12.278,C 0.181,E1 12.4147,E2 481.824} C_DIS
LIN {X 112.908,Y -74.8088,Z 164,A -33.0408,B 12.278,C 0.1815,E1 12.4122,E2 483.4701} C_DIS
LIN {X 110.9514,Y -77.6812,Z 164,A -34.5003,B 12.2779,C 0.1849,E1 12.4099,E2 484.9301} C_DIS
LIN {X 108.917,Y -80.5087,Z 164,A -35.9432,B 12.2779,C 0.1877,E1 12.4075,E2 486.3709} C_DIS
LIN {X 106.5981,Y -83.5541,Z 164,A -37.6477,B 12.2778,C 0.194,E1 12.4046,E2 488.0878} C_DIS
LIN {X 104.0399,Y -86.7197,Z 164,A -39.2647,B 12.2778,C 0.1951,E1 12.4018,E2 489.6938} C_DIS
LIN {X 101.7885,Y -89.3514,Z 164,A -40.716,B 12.2777,C 0.1981,E1 12.3991,E2 491.1451} C_DIS
LIN {X 99.4432,Y -91.9545,Z 164,A -42.2518,B 12.2777,C 0.203,E1 12.3962,E2 492.6892} C_DIS
LIN {X 96.4164,Y -95.1234,Z 164,A -44.0251,B 12.2776,C 0.2048,E1 12.3928,E2 494.4546} C_DIS
LIN {X 93.8947,Y -97.6134,Z 164,A -45.5034,B 12.2776,C 0.2075,E1 12.3898,E2 495.932} C_DIS
LIN {X 91.3372,Y -100.0106,Z 164,A -46.9767,B 12.2775,C 0.2103,E1 12.3868,E2 497.4057} C_DIS
LIN {X 88.4518,Y -102.5705,Z 164,A -48.6766,B 12.2775,C 0.2156,E1 12.3832,E2 499.1158} C_DIS
LIN {X 85.369,Y -105.151,Z 164,A -50.2807,B 12.2774,C 0.2163,E1 12.3798,E2 500.7097} C_DIS
LIN {X 82.6279,Y -107.3183,Z 164,A -51.7467,B 12.2774,C 0.2188,E1 12.3765,E2 502.1758} C_DIS
LIN {X 79.8366,Y -109.4108,Z 164,A -53.2067,B 12.2774,C 0.2211,E1 12.3733,E2 503.6354} C_DIS
LIN {X 76.998,Y -111.4267,Z 164,A -54.6713,B 12.2773,C 0.2235,E1 12.3699,E2 505.1005} C_DIS
LIN {X 74.1153,Y -113.3646,Z 164,A -56.1258,B 12.2773,C 0.2257,E1 12.3665,E2 506.5546} C_DIS
LIN {X 71.2233,Y -115.2033,Z 164,A -57.6659,B 12.2771,C 0.2306,E1 12.3629,E2 508.1074} C_DIS
LIN {X 67.5167,Y -117.4141,Z 164,A -59.5012,B 12.2771,C 0.2338,E1 12.3584,E2 509.9456} C_DIS
LIN {X 63.725,Y -119.5146,Z 164,A -61.2007,B 12.2771,C 0.2329,E1 12.3543,E2 511.6302} C_DIS
LIN {X 60.7495,Y -121.0537,Z 164,A -62.608,B 12.2771,C 0.2347,E1 12.3508,E2 513.0376} C_DIS
LIN {X 57.6827,Y -122.5446,Z 164,A -64.0368,B 12.2771,C 0.2364,E1 12.3472,E2 514.466} C_DIS
LIN {X 54.5264,Y -123.9818,Z 164,A -65.4982,B 12.277,C 0.2382,E1 12.3435,E2 515.928} C_DIS
LIN {X 51.4167,Y -125.3033,Z 164,A -66.9184,B 12.277,C 0.2397,E1 12.3398,E2 517.3483} C_DIS
Enddeposition()
END
